LIN {X 0,Y 536.009,Z 529.66,A -85,B 0,C 180,E1 3996.244,E2 3996.244} C_VEL
LIN {X 0,Y 535.95,Z 529.66,A -85,B 0,C 180,E1 4002.513,E2 4002.513} C_VEL
LIN {X 0,Y 536.324,Z 529.982,A -85,B 0,C 180,E1 4007.164,E2 4007.164} C_VEL
LIN {X 0,Y 539.908,Z 549.024,A -85,B 0,C 180,E1 4007.547,E2 4007.547} C_VEL
LIN {X 0,Y 539.61,Z 624.102,A -85,B 0,C 180,E1 4008.663,E2 4008.663} C_VEL
LIN {X 0,Y 539.026,Z 653.248,A -85,B 0,C 180,E1 4009.753,E2 4009.753} C_VEL
LIN {X 0,Y 538.301,Z 680.399,A -85,B 0,C 180,E1 4011.48,E2 4011.48} C_VEL
LIN {X 0,Y 537.64,Z 703.617,A -85,B 0,C 180,E1 4013.748,E2 4013.748} C_VEL
LIN {X 0,Y 537.126,Z 722.234,A -85,B 0,C 180,E1 4016.46,E2 4016.46} C_VEL
LIN {X 0,Y 536.918,Z 734.161,A -85,B 0,C 180,E1 4019.136,E2 4019.136} C_VEL
LIN {X 0,Y 536.796,Z 741.628,A -85,B 0,C 180,E1 4022.073,E2 4022.073} C_VEL
LIN {X 0,Y 536.618,Z 743.988,A -85,B 0,C 180,E1 4025.051,E2 4025.051} C_VEL
LIN {X 0,Y 536.8,Z 741.206,A -85,B 0,C 180,E1 4028.077,E2 4028.077} C_VEL
LIN {X 0,Y 536.931,Z 732.797,A -85,B 0,C 180,E1 4031.143,E2 4031.143} C_VEL
LIN {X 0,Y 537.282,Z 718.414,A -85,B 0,C 180,E1 4034.107,E2 4034.107} C_VEL
LIN {X 0,Y 537.78,Z 699.357,A -85,B 0,C 180,E1 4036.65,E2 4036.65} C_VEL
LIN {X 0,Y 538.453,Z 675.808,A -85,B 0,C 180,E1 4038.779,E2 4038.779} C_VEL
LIN {X 0,Y 539.118,Z 648.555,A -85,B 0,C 180,E1 4040.382,E2 4040.382} C_VEL
LIN {X 0,Y 539.716,Z 619.376,A -85,B 0,C 180,E1 4041.356,E2 4041.356} C_VEL
LIN {X 0,Y 539.014,Z 540.519,A -85,B 0,C 180,E1 4042.509,E2 4042.509} C_VEL
LIN {X 0,Y 536.185,Z 529.66,A -85,B 0,C 180,E1 4042.825,E2 4042.825} C_VEL
LIN {X 0,Y 536.413,Z 529.66,A -85,B 0,C 180,E1 4048.387,E2 4048.387} C_VEL
LIN {X 0,Y 536.478,Z 529.66,A -85,B 0,C 180,E1 4053.224,E2 4053.224} C_VEL
LIN {X 0,Y 536.337,Z 529.66,A -85,B 0,C 180,E1 4058.086,E2 4058.086} C_VEL
LIN {X 0,Y 536.259,Z 529.66,A -85,B 0,C 180,E1 4063.009,E2 4063.009} C_VEL
LIN {X 0,Y 536.257,Z 529.66,A -85,B 0,C 180,E1 4068.03,E2 4068.03} C_VEL
LIN {X 0,Y 536.18,Z 529.66,A -85,B 0,C 180,E1 4073.203,E2 4073.203} C_VEL
LIN {X 0,Y 535.995,Z 529.66,A -85,B 0,C 180,E1 4079.218,E2 4079.218} C_VEL
LIN {X 0,Y 536.078,Z 529.66,A -85,B 0,C 180,E1 4085.28,E2 4085.28} C_VEL
LIN {X 0,Y 536.058,Z 529.66,A -85,B 0,C 180,E1 4090.53,E2 4090.53} C_VEL
LIN {X 0,Y 536.047,Z 529.66,A -85,B 0,C 180,E1 4097.046,E2 4097.046} C_VEL
LIN {X 0,Y 536.127,Z 529.66,A -85,B 0,C 180,E1 4102.006,E2 4102.006} C_VEL
LIN {X 0,Y 536.002,Z 529.66,A -85,B 0,C 180,E1 4107.661,E2 4107.661} C_VEL
LIN {X 0,Y 536.225,Z 529.66,A -85,B 0,C 180,E1 4114.224,E2 4114.224} C_VEL
LIN {X 0,Y 536.413,Z 529.66,A -85,B 0,C 180,E1 4115.573,E2 4115.573} C_VEL
LIN {X 0,Y 542.639,Z 549.532,A -85,B 0,C 180,E1 4116.157,E2 4116.157} C_VEL
LIN {X 0,Y 542.031,Z 585.577,A -85,B 0,C 180,E1 4116.981,E2 4116.981} C_VEL
LIN {X 0,Y 540.981,Z 619.2,A -85,B 0,C 180,E1 4118.415,E2 4118.415} C_VEL
LIN {X 0,Y 539.732,Z 651.158,A -85,B 0,C 180,E1 4120.501,E2 4120.501} C_VEL
LIN {X 0,Y 538.579,Z 677.691,A -85,B 0,C 180,E1 4122.945,E2 4122.945} C_VEL
LIN {X 0,Y 537.718,Z 701.766,A -85,B 0,C 180,E1 4125.994,E2 4125.994} C_VEL
LIN {X 0,Y 537.159,Z 719.995,A -85,B 0,C 180,E1 4129.228,E2 4129.228} C_VEL
LIN {X 0,Y 536.883,Z 733.409,A -85,B 0,C 180,E1 4132.732,E2 4132.732} C_VEL
LIN {X 0,Y 536.795,Z 740.394,A -85,B 0,C 180,E1 4135.732,E2 4135.732} C_VEL
LIN {X 0,Y 536.721,Z 743.474,A -85,B 0,C 180,E1 4138.387,E2 4138.387} C_VEL
LIN {X 0,Y 536.852,Z 743.419,A -85,B 0,C 180,E1 4141.609,E2 4141.609} C_VEL
LIN {X 0,Y 536.807,Z 739.198,A -85,B 0,C 180,E1 4144.835,E2 4144.835} C_VEL
LIN {X 0,Y 536.965,Z 729.095,A -85,B 0,C 180,E1 4148.482,E2 4148.482} C_VEL
LIN {X 0,Y 537.316,Z 713.592,A -85,B 0,C 180,E1 4151.951,E2 4151.951} C_VEL
LIN {X 0,Y 538.008,Z 693.827,A -85,B 0,C 180,E1 4155.035,E2 4155.035} C_VEL
LIN {X 0,Y 538.992,Z 668.188,A -85,B 0,C 180,E1 4157.934,E2 4157.934} C_VEL
LIN {X 0,Y 540.269,Z 638.35,A -85,B 0,C 180,E1 4160.343,E2 4160.343} C_VEL
LIN {X 0,Y 541.151,Z 614.891,A -85,B 0,C 180,E1 4161.718,E2 4161.718} C_VEL
LIN {X 0,Y 537.972,Z 599.622,A -85,B 0,C 180,E1 4162.578,E2 4162.578} C_VEL
LIN {X 0,Y 534.792,Z 585.979,A -85,B 0,C 180,E1 4163.245,E2 4163.245} C_VEL
LIN {X 0,Y 534.777,Z 583.899,A -85,B 0,C 180,E1 4163.316,E2 4163.316} C_VEL
LIN {X 0,Y 534.711,Z 547.853,A -85,B 0,C 180,E1 4164.152,E2 4164.152} C_VEL
LIN {X 0,Y 528.282,Z 529.66,A -85,B 0,C 180,E1 4164.754,E2 4164.754} C_VEL
LIN {X 0,Y 528.142,Z 529.66,A -85,B 0,C 180,E1 4171.003,E2 4171.003} C_VEL
LIN {X 0,Y 528.088,Z 529.66,A -85,B 0,C 180,E1 4176.871,E2 4176.871} C_VEL
LIN {X 0,Y 527.998,Z 529.66,A -85,B 0,C 180,E1 4183.303,E2 4183.303} C_VEL
LIN {X 0,Y 528.131,Z 529.66,A -85,B 0,C 180,E1 4188.917,E2 4188.917} C_VEL
LIN {X 0,Y 528.135,Z 529.66,A -85,B 0,C 180,E1 4195.15,E2 4195.15} C_VEL
LIN {X 0,Y 528.223,Z 529.66,A -85,B 0,C 180,E1 4200.411,E2 4200.411} C_VEL
LIN {X 0,Y 537.906,Z 555.81,A -85,B 0,C 180,E1 4201.345,E2 4201.345} C_VEL
LIN {X 0,Y 537.262,Z 596.398,A -85,B 0,C 180,E1 4202.129,E2 4202.129} C_VEL
LIN {X 0,Y 535.972,Z 632.816,A -85,B 0,C 180,E1 4203.464,E2 4203.464} C_VEL
LIN {X 0,Y 534.3,Z 668.478,A -85,B 0,C 180,E1 4205.493,E2 4205.493} C_VEL
LIN {X 0,Y 532.62,Z 699.844,A -85,B 0,C 180,E1 4208.007,E2 4208.007} C_VEL
LIN {X 0,Y 531.125,Z 727.043,A -85,B 0,C 180,E1 4210.93,E2 4210.93} C_VEL
LIN {X 0,Y 529.939,Z 751.815,A -85,B 0,C 180,E1 4214.518,E2 4214.518} C_VEL
LIN {X 0,Y 529.276,Z 769.655,A -85,B 0,C 180,E1 4218.072,E2 4218.072} C_VEL
LIN {X 0,Y 528.98,Z 782.685,A -85,B 0,C 180,E1 4221.801,E2 4221.801} C_VEL
LIN {X 0,Y 528.862,Z 791.191,A -85,B 0,C 180,E1 4225.91,E2 4225.91} C_VEL
LIN {X 0,Y 528.783,Z 794,A -85,B 0,C 180,E1 4230.001,E2 4230.001} C_VEL
LIN {X 0,Y 528.901,Z 791.19,A -85,B 0,C 180,E1 4234.091,E2 4234.091} C_VEL
LIN {X 0,Y 529.004,Z 782.678,A -85,B 0,C 180,E1 4238.201,E2 4238.201} C_VEL
LIN {X 0,Y 529.253,Z 769.649,A -85,B 0,C 180,E1 4241.93,E2 4241.93} C_VEL
LIN {X 0,Y 529.975,Z 750.599,A -85,B 0,C 180,E1 4245.694,E2 4245.694} C_VEL
LIN {X 0,Y 531.118,Z 727.031,A -85,B 0,C 180,E1 4249.071,E2 4249.071} C_VEL
LIN {X 0,Y 532.597,Z 699.86,A -85,B 0,C 180,E1 4251.992,E2 4251.992} C_VEL
LIN {X 0,Y 534.276,Z 668.46,A -85,B 0,C 180,E1 4254.509,E2 4254.509} C_VEL
LIN {X 0,Y 535.917,Z 633.307,A -85,B 0,C 180,E1 4256.516,E2 4256.516} C_VEL
LIN {X 0,Y 537.203,Z 596.71,A -85,B 0,C 180,E1 4257.866,E2 4257.866} C_VEL
LIN {X 0,Y 537.47,Z 553.409,A -85,B 0,C 180,E1 4258.717,E2 4258.717} C_VEL
LIN {X 0,Y 528.217,Z 529.66,A -85,B 0,C 180,E1 4259.593,E2 4259.593} C_VEL
LIN {X 0,Y 528.124,Z 529.66,A -85,B 0,C 180,E1 4264.852,E2 4264.852} C_VEL
LIN {X 0,Y 528.156,Z 529.66,A -85,B 0,C 180,E1 4269.523,E2 4269.523} C_VEL
LIN {X 0,Y 528.089,Z 529.66,A -85,B 0,C 180,E1 4275.592,E2 4275.592} C_VEL
LIN {X 0,Y 528.134,Z 529.66,A -85,B 0,C 180,E1 4281.057,E2 4281.057} C_VEL
LIN {X 0,Y 528.12,Z 529.66,A -85,B 0,C 180,E1 4287.123,E2 4287.123} C_VEL
LIN {X 0,Y 528.196,Z 529.66,A -85,B 0,C 180,E1 4292.803,E2 4292.803} C_VEL
LIN {X 0,Y 528.328,Z 529.66,A -85,B 0,C 180,E1 4298.207,E2 4298.207} C_VEL
LIN {X 0,Y 528.423,Z 529.66,A -85,B 0,C 180,E1 4303.41,E2 4303.41} C_VEL
LIN {X 0,Y 528.47,Z 529.66,A -85,B 0,C 180,E1 4310.138,E2 4310.138} C_VEL
LIN {X 0,Y 528.582,Z 529.66,A -85,B 0,C 180,E1 4315.089,E2 4315.089} C_VEL
LIN {X 0,Y 528.64,Z 529.66,A -85,B 0,C 180,E1 4320.002,E2 4320.002} C_VEL
LIN {X 0,Y 528.61,Z 529.66,A -85,B 0,C 180,E1 4324.915,E2 4324.915} C_VEL
LIN {X 0,Y 528.501,Z 529.66,A -85,B 0,C 180,E1 4329.866,E2 4329.866} C_VEL
LIN {X 0,Y 528.464,Z 529.66,A -85,B 0,C 180,E1 4334.894,E2 4334.894} C_VEL
LIN {X 0,Y 528.375,Z 529.66,A -85,B 0,C 180,E1 4340.044,E2 4340.044} C_VEL
LIN {X 0,Y 528.202,Z 529.66,A -85,B 0,C 180,E1 4345.376,E2 4345.376} C_VEL
LIN {X 0,Y 528.141,Z 529.66,A -85,B 0,C 180,E1 4351,E2 4351} C_VEL
LIN {X 0,Y 528.069,Z 529.66,A -85,B 0,C 180,E1 4356.878,E2 4356.878} C_VEL
LIN {X 0,Y 528.014,Z 529.66,A -85,B 0,C 180,E1 4363.308,E2 4363.308} C_VEL
LIN {X 0,Y 528.365,Z 529.66,A -85,B 0,C 180,E1 4366.859,E2 4366.859} C_VEL
LIN {X 0,Y 532.147,Z 547.399,A -85,B 0,C 180,E1 4367.261,E2 4367.261} C_VEL
LIN {X 0,Y 532.046,Z 624.585,A -85,B 0,C 180,E1 4368.431,E2 4368.431} C_VEL
LIN {X 0,Y 531.393,Z 653.619,A -85,B 0,C 180,E1 4369.532,E2 4369.532} C_VEL
LIN {X 0,Y 530.6,Z 680.452,A -85,B 0,C 180,E1 4371.268,E2 4371.268} C_VEL
LIN {X 0,Y 529.858,Z 702.607,A -85,B 0,C 180,E1 4373.452,E2 4373.452} C_VEL
LIN {X 0,Y 529.328,Z 720.972,A -85,B 0,C 180,E1 4376.111,E2 4376.111} C_VEL
LIN {X 0,Y 529.026,Z 734.353,A -85,B 0,C 180,E1 4379.107,E2 4379.107} C_VEL
LIN {X 0,Y 528.89,Z 741.859,A -85,B 0,C 180,E1 4382.19,E2 4382.19} C_VEL
LIN {X 0,Y 528.738,Z 743.945,A -85,B 0,C 180,E1 4384.653,E2 4384.653} C_VEL
LIN {X 0,Y 528.842,Z 741.854,A -85,B 0,C 180,E1 4387.729,E2 4387.729} C_VEL
LIN {X 0,Y 529.034,Z 734.88,A -85,B 0,C 180,E1 4390.639,E2 4390.639} C_VEL
LIN {X 0,Y 529.289,Z 721.837,A -85,B 0,C 180,E1 4393.647,E2 4393.647} C_VEL
LIN {X 0,Y 529.88,Z 703.234,A -85,B 0,C 180,E1 4396.38,E2 4396.38} C_VEL
LIN {X 0,Y 530.598,Z 680.819,A -85,B 0,C 180,E1 4398.611,E2 4398.611} C_VEL
LIN {X 0,Y 531.409,Z 654.236,A -85,B 0,C 180,E1 4400.344,E2 4400.344} C_VEL
LIN {X 0,Y 531.994,Z 626.187,A -85,B 0,C 180,E1 4401.435,E2 4401.435} C_VEL
LIN {X 0,Y 532.245,Z 567.67,A -85,B 0,C 180,E1 4402.364,E2 4402.364} C_VEL
LIN {X 0,Y 531.319,Z 541.394,A -85,B 0,C 180,E1 4402.761,E2 4402.761} C_VEL
LIN {X 0,Y 528.288,Z 529.66,A -85,B 0,C 180,E1 4403.116,E2 4403.116} C_VEL
LIN {X 0,Y 528.523,Z 529.66,A -85,B 0,C 180,E1 4408.363,E2 4408.363} C_VEL
LIN {X 0,Y 528.585,Z 529.66,A -85,B 0,C 180,E1 4413.272,E2 4413.272} C_VEL
LIN {X 0,Y 528.44,Z 529.66,A -85,B 0,C 180,E1 4418.208,E2 4418.208} C_VEL
LIN {X 0,Y 528.313,Z 529.66,A -85,B 0,C 180,E1 4423.797,E2 4423.797} C_VEL
LIN {X 0,Y 528.374,Z 529.66,A -85,B 0,C 180,E1 4429.528,E2 4429.528} C_VEL
LIN {X 0,Y 528.205,Z 529.66,A -85,B 0,C 180,E1 4435.373,E2 4435.373} C_VEL
LIN {X 0,Y 528.09,Z 529.66,A -85,B 0,C 180,E1 4440.989,E2 4440.989} C_VEL
LIN {X 0,Y 528.255,Z 529.66,A -85,B 0,C 180,E1 4446.883,E2 4446.883} C_VEL
LIN {X 0,Y 528.03,Z 529.66,A -85,B 0,C 180,E1 4453.303,E2 4453.303} C_VEL
LIN {X 0,Y 528.103,Z 529.66,A -85,B 0,C 180,E1 4458.911,E2 4458.911} C_VEL
LIN {X 0,Y 528.069,Z 529.66,A -85,B 0,C 180,E1 4465.142,E2 4465.142} C_VEL
LIN {X 0,Y 528.155,Z 529.66,A -85,B 0,C 180,E1 4470.939,E2 4470.939} C_VEL
LIN {X 0,Y 528.447,Z 529.66,A -85,B 0,C 180,E1 4475.163,E2 4475.163} C_VEL
LIN {X 0,Y 535.451,Z 551.381,A -85,B 0,C 180,E1 4475.846,E2 4475.846} C_VEL
LIN {X 0,Y 534.695,Z 586.678,A -85,B 0,C 180,E1 4476.686,E2 4476.686} C_VEL
LIN {X 0,Y 533.505,Z 621.104,A -85,B 0,C 180,E1 4478.206,E2 4478.206} C_VEL
LIN {X 0,Y 532.146,Z 652.485,A -85,B 0,C 180,E1 4480.32,E2 4480.32} C_VEL
LIN {X 0,Y 530.818,Z 680.078,A -85,B 0,C 180,E1 4482.955,E2 4482.955} C_VEL
LIN {X 0,Y 529.842,Z 704.046,A -85,B 0,C 180,E1 4486.136,E2 4486.136} C_VEL
LIN {X 0,Y 529.258,Z 721.344,A -85,B 0,C 180,E1 4489.356,E2 4489.356} C_VEL
LIN {X 0,Y 528.995,Z 734.551,A -85,B 0,C 180,E1 4493.035,E2 4493.035} C_VEL
LIN {X 0,Y 528.917,Z 741.947,A -85,B 0,C 180,E1 4496.727,E2 4496.727} C_VEL
LIN {X 0,Y 528.806,Z 743.997,A -85,B 0,C 180,E1 4499.998,E2 4499.998} C_VEL
LIN {X 0,Y 528.916,Z 741.843,A -85,B 0,C 180,E1 4503.269,E2 4503.269} C_VEL
LIN {X 0,Y 529.011,Z 734.311,A -85,B 0,C 180,E1 4506.961,E2 4506.961} C_VEL
LIN {X 0,Y 529.356,Z 720.626,A -85,B 0,C 180,E1 4510.708,E2 4510.708} C_VEL
LIN {X 0,Y 530.015,Z 701.179,A -85,B 0,C 180,E1 4514.211,E2 4514.211} C_VEL
LIN {X 0,Y 530.959,Z 677.649,A -85,B 0,C 180,E1 4517.221,E2 4517.221} C_VEL
LIN {X 0,Y 532.276,Z 650.083,A -85,B 0,C 180,E1 4519.778,E2 4519.778} C_VEL
LIN {X 0,Y 533.553,Z 619.596,A -85,B 0,C 180,E1 4521.787,E2 4521.787} C_VEL
LIN {X 0,Y 534.723,Z 585.396,A -85,B 0,C 180,E1 4523.268,E2 4523.268} C_VEL
LIN {X 0,Y 534.777,Z 583.899,A -85,B 0,C 180,E1 4523.316,E2 4523.316} C_VEL
LIN {X 0,Y 533.025,Z 567.224,A -85,B 0,C 180,E1 4523.874,E2 4523.874} C_VEL
LIN {X 0,Y 527.988,Z 551.07,A -85,B 0,C 180,E1 4524.432,E2 4524.432} C_VEL
LIN {X 0,Y 520.329,Z 529.66,A -85,B 0,C 180,E1 4525.219,E2 4525.219} C_VEL
LIN {X 0,Y 520.224,Z 529.66,A -85,B 0,C 180,E1 4531.471,E2 4531.471} C_VEL
LIN {X 0,Y 520.089,Z 529.66,A -85,B 0,C 180,E1 4537.535,E2 4537.535} C_VEL
LIN {X 0,Y 520.093,Z 529.66,A -85,B 0,C 180,E1 4543.503,E2 4543.503} C_VEL
LIN {X 0,Y 520.228,Z 529.66,A -85,B 0,C 180,E1 4548.948,E2 4548.948} C_VEL
LIN {X 0,Y 520.185,Z 529.66,A -85,B 0,C 180,E1 4554.538,E2 4554.538} C_VEL
LIN {X 0,Y 520.314,Z 529.66,A -85,B 0,C 180,E1 4560.082,E2 4560.082} C_VEL
LIN {X 0,Y 530.949,Z 556.615,A -85,B 0,C 180,E1 4560.953,E2 4560.953} C_VEL
LIN {X 0,Y 530.248,Z 597.126,A -85,B 0,C 180,E1 4561.748,E2 4561.748} C_VEL
LIN {X 0,Y 528.822,Z 632.931,A -85,B 0,C 180,E1 4563.082,E2 4563.082} C_VEL
LIN {X 0,Y 526.98,Z 668.474,A -85,B 0,C 180,E1 4565.13,E2 4565.13} C_VEL
LIN {X 0,Y 525.142,Z 700.197,A -85,B 0,C 180,E1 4567.712,E2 4567.712} C_VEL
LIN {X 0,Y 523.41,Z 728.787,A -85,B 0,C 180,E1 4570.857,E2 4570.857} C_VEL
LIN {X 0,Y 522.103,Z 753.018,A -85,B 0,C 180,E1 4574.494,E2 4574.494} C_VEL
LIN {X 0,Y 521.367,Z 771.385,A -85,B 0,C 180,E1 4578.312,E2 4578.312} C_VEL
LIN {X 0,Y 521.057,Z 783.828,A -85,B 0,C 180,E1 4582.094,E2 4582.094} C_VEL
LIN {X 0,Y 520.959,Z 791.192,A -85,B 0,C 180,E1 4585.848,E2 4585.848} C_VEL
LIN {X 0,Y 520.889,Z 794,A -85,B 0,C 180,E1 4590.001,E2 4590.001} C_VEL
LIN {X 0,Y 520.994,Z 791.191,A -85,B 0,C 180,E1 4594.153,E2 4594.153} C_VEL
LIN {X 0,Y 521.115,Z 782.678,A -85,B 0,C 180,E1 4598.326,E2 4598.326} C_VEL
LIN {X 0,Y 521.409,Z 769.649,A -85,B 0,C 180,E1 4602.113,E2 4602.113} C_VEL
LIN {X 0,Y 522.207,Z 750.6,A -85,B 0,C 180,E1 4605.934,E2 4605.934} C_VEL
LIN {X 0,Y 523.475,Z 727.031,A -85,B 0,C 180,E1 4609.361,E2 4609.361} C_VEL
LIN {X 0,Y 525.23,Z 698.46,A -85,B 0,C 180,E1 4612.453,E2 4612.453} C_VEL
LIN {X 0,Y 527.094,Z 666.926,A -85,B 0,C 180,E1 4614.979,E2 4614.979} C_VEL
LIN {X 0,Y 528.927,Z 631.177,A -85,B 0,C 180,E1 4616.995,E2 4616.995} C_VEL
LIN {X 0,Y 530.246,Z 596.382,A -85,B 0,C 180,E1 4618.273,E2 4618.273} C_VEL
LIN {X 0,Y 530.592,Z 555.708,A -85,B 0,C 180,E1 4619.079,E2 4619.079} C_VEL
LIN {X 0,Y 520.275,Z 529.66,A -85,B 0,C 180,E1 4620.061,E2 4620.061} C_VEL
LIN {X 0,Y 520.216,Z 529.66,A -85,B 0,C 180,E1 4625.694,E2 4625.694} C_VEL
LIN {X 0,Y 520.191,Z 529.66,A -85,B 0,C 180,E1 4631.047,E2 4631.047} C_VEL
LIN {X 0,Y 520.173,Z 529.66,A -85,B 0,C 180,E1 4636.489,E2 4636.489} C_VEL
LIN {X 0,Y 520.224,Z 529.66,A -85,B 0,C 180,E1 4642.476,E2 4642.476} C_VEL
LIN {X 0,Y 520.192,Z 529.66,A -85,B 0,C 180,E1 4648.526,E2 4648.526} C_VEL
LIN {X 0,Y 520.295,Z 529.66,A -85,B 0,C 180,E1 4654.215,E2 4654.215} C_VEL
LIN {X 0,Y 520.449,Z 529.66,A -85,B 0,C 180,E1 4659.642,E2 4659.642} C_VEL
LIN {X 0,Y 520.358,Z 529.66,A -85,B 0,C 180,E1 4664.874,E2 4664.874} C_VEL
LIN {X 0,Y 520.585,Z 529.66,A -85,B 0,C 180,E1 4670.248,E2 4670.248} C_VEL
LIN {X 0,Y 520.677,Z 529.66,A -85,B 0,C 180,E1 4675.014,E2 4675.014} C_VEL
LIN {X 0,Y 520.752,Z 529.66,A -85,B 0,C 180,E1 4680.002,E2 4680.002} C_VEL
LIN {X 0,Y 520.695,Z 529.66,A -85,B 0,C 180,E1 4684.99,E2 4684.99} C_VEL
LIN {X 0,Y 520.576,Z 529.66,A -85,B 0,C 180,E1 4690.018,E2 4690.018} C_VEL
LIN {X 0,Y 520.53,Z 529.66,A -85,B 0,C 180,E1 4695.126,E2 4695.126} C_VEL
LIN {X 0,Y 520.431,Z 529.66,A -85,B 0,C 180,E1 4700.363,E2 4700.363} C_VEL
LIN {X 0,Y 520.236,Z 529.66,A -85,B 0,C 180,E1 4705.948,E2 4705.948} C_VEL
LIN {X 0,Y 520.212,Z 529.66,A -85,B 0,C 180,E1 4711.477,E2 4711.477} C_VEL
LIN {X 0,Y 520.063,Z 529.66,A -85,B 0,C 180,E1 4717.543,E2 4717.543} C_VEL
LIN {X 0,Y 520.112,Z 529.66,A -85,B 0,C 180,E1 4723.503,E2 4723.503} C_VEL
LIN {X 0,Y 520.402,Z 529.66,A -85,B 0,C 180,E1 4726.575,E2 4726.575} C_VEL
LIN {X 0,Y 524.617,Z 548.131,A -85,B 0,C 180,E1 4727.007,E2 4727.007} C_VEL
LIN {X 0,Y 524.49,Z 625.285,A -85,B 0,C 180,E1 4728.198,E2 4728.198} C_VEL
LIN {X 0,Y 523.813,Z 653.189,A -85,B 0,C 180,E1 4729.263,E2 4729.263} C_VEL
LIN {X 0,Y 522.986,Z 679.327,A -85,B 0,C 180,E1 4730.947,E2 4730.947} C_VEL
LIN {X 0,Y 522.129,Z 702.433,A -85,B 0,C 180,E1 4733.211,E2 4733.211} C_VEL
LIN {X 0,Y 521.522,Z 721.035,A -85,B 0,C 180,E1 4735.943,E2 4735.943} C_VEL
LIN {X 0,Y 521.159,Z 734.536,A -85,B 0,C 180,E1 4739.042,E2 4739.042} C_VEL
LIN {X 0,Y 520.978,Z 742.239,A -85,B 0,C 180,E1 4742.39,E2 4742.39} C_VEL
LIN {X 0,Y 520.814,Z 743.86,A -85,B 0,C 180,E1 4744.239,E2 4744.239} C_VEL
LIN {X 0,Y 520.823,Z 743.638,A -85,B 0,C 180,E1 4746.069,E2 4746.069} C_VEL
LIN {X 0,Y 521.069,Z 740.017,A -85,B 0,C 180,E1 4748.815,E2 4748.815} C_VEL
LIN {X 0,Y 521.235,Z 731.187,A -85,B 0,C 180,E1 4751.796,E2 4751.796} C_VEL
LIN {X 0,Y 521.667,Z 716.778,A -85,B 0,C 180,E1 4754.695,E2 4754.695} C_VEL
LIN {X 0,Y 522.31,Z 697.392,A -85,B 0,C 180,E1 4757.273,E2 4757.273} C_VEL
LIN {X 0,Y 523.161,Z 674.318,A -85,B 0,C 180,E1 4759.345,E2 4759.345} C_VEL
LIN {X 0,Y 523.975,Z 647.028,A -85,B 0,C 180,E1 4760.938,E2 4760.938} C_VEL
LIN {X 0,Y 524.556,Z 617.97,A -85,B 0,C 180,E1 4761.886,E2 4761.886} C_VEL
LIN {X 0,Y 523.89,Z 543.047,A -85,B 0,C 180,E1 4763,E2 4763} C_VEL
LIN {X 0,Y 520.363,Z 529.66,A -85,B 0,C 180,E1 4763.338,E2 4763.338} C_VEL
LIN {X 0,Y 520.647,Z 529.66,A -85,B 0,C 180,E1 4768.338,E2 4768.338} C_VEL
LIN {X 0,Y 520.681,Z 529.66,A -85,B 0,C 180,E1 4773.322,E2 4773.322} C_VEL
LIN {X 0,Y 520.528,Z 529.66,A -85,B 0,C 180,E1 4778.334,E2 4778.334} C_VEL
LIN {X 0,Y 520.452,Z 529.66,A -85,B 0,C 180,E1 4783.411,E2 4783.411} C_VEL
LIN {X 0,Y 520.433,Z 529.66,A -85,B 0,C 180,E1 4788.598,E2 4788.598} C_VEL
LIN {X 0,Y 520.314,Z 529.66,A -85,B 0,C 180,E1 4793.954,E2 4793.954} C_VEL
LIN {X 0,Y 520.179,Z 529.66,A -85,B 0,C 180,E1 4799.547,E2 4799.547} C_VEL
LIN {X 0,Y 520.231,Z 529.66,A -85,B 0,C 180,E1 4805.688,E2 4805.688} C_VEL
LIN {X 0,Y 520.168,Z 529.66,A -85,B 0,C 180,E1 4811.037,E2 4811.037} C_VEL
LIN {X 0,Y 520.184,Z 529.66,A -85,B 0,C 180,E1 4816.486,E2 4816.486} C_VEL
LIN {X 0,Y 520.171,Z 529.66,A -85,B 0,C 180,E1 4822.466,E2 4822.466} C_VEL
LIN {X 0,Y 520.164,Z 529.66,A -85,B 0,C 180,E1 4828.519,E2 4828.519} C_VEL
LIN {X 0,Y 520.475,Z 529.66,A -85,B 0,C 180,E1 4834.777,E2 4834.777} C_VEL
LIN {X 0,Y 528.239,Z 553.901,A -85,B 0,C 180,E1 4835.538,E2 4835.538} C_VEL
LIN {X 0,Y 527.355,Z 589.315,A -85,B 0,C 180,E1 4836.439,E2 4836.439} C_VEL
LIN {X 0,Y 526.049,Z 623.008,A -85,B 0,C 180,E1 4837.992,E2 4837.992} C_VEL
LIN {X 0,Y 524.544,Z 653.801,A -85,B 0,C 180,E1 4840.132,E2 4840.132} C_VEL
LIN {X 0,Y 523.068,Z 682.108,A -85,B 0,C 180,E1 4842.927,E2 4842.927} C_VEL
LIN {X 0,Y 522.05,Z 704.573,A -85,B 0,C 180,E1 4846.01,E2 4846.01} C_VEL
LIN {X 0,Y 521.357,Z 722.985,A -85,B 0,C 180,E1 4849.587,E2 4849.587} C_VEL
LIN {X 0,Y 521.127,Z 734.55,A -85,B 0,C 180,E1 4852.929,E2 4852.929} C_VEL
LIN {X 0,Y 521.014,Z 741.943,A -85,B 0,C 180,E1 4856.677,E2 4856.677} C_VEL
LIN {X 0,Y 520.912,Z 743.997,A -85,B 0,C 180,E1 4859.998,E2 4859.998} C_VEL
LIN {X 0,Y 521.014,Z 741.841,A -85,B 0,C 180,E1 4863.318,E2 4863.318} C_VEL
LIN {X 0,Y 521.147,Z 734.314,A -85,B 0,C 180,E1 4867.066,E2 4867.066} C_VEL
LIN {X 0,Y 521.516,Z 720.605,A -85,B 0,C 180,E1 4870.877,E2 4870.877} C_VEL
LIN {X 0,Y 522.228,Z 701.986,A -85,B 0,C 180,E1 4874.306,E2 4874.306} C_VEL
LIN {X 0,Y 523.249,Z 678.576,A -85,B 0,C 180,E1 4877.379,E2 4877.379} C_VEL
LIN {X 0,Y 524.676,Z 651.439,A -85,B 0,C 180,E1 4879.968,E2 4879.968} C_VEL
LIN {X 0,Y 526.176,Z 619.604,A -85,B 0,C 180,E1 4882.108,E2 4882.108} C_VEL
LIN {X 0,Y 527.456,Z 585.415,A -85,B 0,C 180,E1 4883.608,E2 4883.608} C_VEL
LIN {X 0,Y 527.988,Z 551.07,A -85,B 0,C 180,E1 4884.432,E2 4884.432} C_VEL
LIN {X 0,Y 520.994,Z 542.646,A -85,B 0,C 180,E1 4884.915,E2 4884.915} C_VEL
LIN {X 0,Y 513.747,Z 534.323,A -85,B 0,C 180,E1 4885.406,E2 4885.406} C_VEL
LIN {X 0,Y 512.392,Z 529.66,A -85,B 0,C 180,E1 4885.606,E2 4885.606} C_VEL
LIN {X 0,Y 512.331,Z 529.66,A -85,B 0,C 180,E1 4892.013,E2 4892.013} C_VEL
LIN {X 0,Y 512.185,Z 529.66,A -85,B 0,C 180,E1 4898.218,E2 4898.218} C_VEL
LIN {X 0,Y 512.196,Z 529.66,A -85,B 0,C 180,E1 4905.004,E2 4905.004} C_VEL
LIN {X 0,Y 512.323,Z 529.66,A -85,B 0,C 180,E1 4909.974,E2 4909.974} C_VEL
LIN {X 0,Y 512.241,Z 529.66,A -85,B 0,C 180,E1 4915.965,E2 4915.965} C_VEL
LIN {X 0,Y 512.368,Z 529.66,A -85,B 0,C 180,E1 4919.726,E2 4919.726} C_VEL
LIN {X 0,Y 523.614,Z 558.863,A -85,B 0,C 180,E1 4920.666,E2 4920.666} C_VEL
LIN {X 0,Y 522.963,Z 599.981,A -85,B 0,C 180,E1 4921.483,E2 4921.483} C_VEL
LIN {X 0,Y 521.555,Z 636.941,A -85,B 0,C 180,E1 4922.891,E2 4922.891} C_VEL
LIN {X 0,Y 519.617,Z 670.002,A -85,B 0,C 180,E1 4924.868,E2 4924.868} C_VEL
LIN {X 0,Y 517.639,Z 700.696,A -85,B 0,C 180,E1 4927.42,E2 4927.42} C_VEL
LIN {X 0,Y 515.791,Z 728.787,A -85,B 0,C 180,E1 4930.563,E2 4930.563} C_VEL
LIN {X 0,Y 514.357,Z 753.017,A -85,B 0,C 180,E1 4934.255,E2 4934.255} C_VEL
LIN {X 0,Y 513.523,Z 771.385,A -85,B 0,C 180,E1 4938.131,E2 4938.131} C_VEL
LIN {X 0,Y 513.197,Z 783.828,A -85,B 0,C 180,E1 4941.972,E2 4941.972} C_VEL
LIN {X 0,Y 513.057,Z 791.192,A -85,B 0,C 180,E1 4945.784,E2 4945.784} C_VEL
LIN {X 0,Y 512.994,Z 794,A -85,B 0,C 180,E1 4950.001,E2 4950.001} C_VEL
LIN {X 0,Y 513.087,Z 791.191,A -85,B 0,C 180,E1 4954.217,E2 4954.217} C_VEL
LIN {X 0,Y 513.245,Z 782.678,A -85,B 0,C 180,E1 4958.454,E2 4958.454} C_VEL
LIN {X 0,Y 513.561,Z 769.648,A -85,B 0,C 180,E1 4962.3,E2 4962.3} C_VEL
LIN {X 0,Y 514.456,Z 750.601,A -85,B 0,C 180,E1 4966.18,E2 4966.18} C_VEL
LIN {X 0,Y 515.853,Z 727.03,A -85,B 0,C 180,E1 4969.659,E2 4969.659} C_VEL
LIN {X 0,Y 517.708,Z 699.2,A -85,B 0,C 180,E1 4972.724,E2 4972.724} C_VEL
LIN {X 0,Y 519.823,Z 666.922,A -85,B 0,C 180,E1 4975.353,E2 4975.353} C_VEL
LIN {X 0,Y 521.766,Z 632.261,A -85,B 0,C 180,E1 4977.331,E2 4977.331} C_VEL
LIN {X 0,Y 523.111,Z 596.014,A -85,B 0,C 180,E1 4978.651,E2 4978.651} C_VEL
LIN {X 0,Y 523.218,Z 557.302,A -85,B 0,C 180,E1 4979.433,E2 4979.433} C_VEL
LIN {X 0,Y 512.35,Z 529.66,A -85,B 0,C 180,E1 4980.517,E2 4980.517} C_VEL
LIN {X 0,Y 512.337,Z 529.66,A -85,B 0,C 180,E1 4987.327,E2 4987.327} C_VEL
LIN {X 0,Y 512.18,Z 529.66,A -85,B 0,C 180,E1 4992.66,E2 4992.66} C_VEL
LIN {X 0,Y 512.246,Z 529.66,A -85,B 0,C 180,E1 4997.432,E2 4997.432} C_VEL
LIN {X 0,Y 512.294,Z 529.66,A -85,B 0,C 180,E1 5002.685,E2 5002.685} C_VEL
LIN {X 0,Y 512.29,Z 529.66,A -85,B 0,C 180,E1 5008.675,E2 5008.675} C_VEL
LIN {X 0,Y 512.366,Z 529.66,A -85,B 0,C 180,E1 5013.786,E2 5013.786} C_VEL
LIN {X 0,Y 512.541,Z 529.66,A -85,B 0,C 180,E1 5019.314,E2 5019.314} C_VEL
LIN {X 0,Y 512.451,Z 529.66,A -85,B 0,C 180,E1 5024.634,E2 5024.634} C_VEL
LIN {X 0,Y 512.625,Z 529.66,A -85,B 0,C 180,E1 5029.83,E2 5029.83} C_VEL
LIN {X 0,Y 512.796,Z 529.66,A -85,B 0,C 180,E1 5034.938,E2 5034.938} C_VEL
LIN {X 0,Y 512.858,Z 529.66,A -85,B 0,C 180,E1 5040.002,E2 5040.002} C_VEL
LIN {X 0,Y 512.806,Z 529.66,A -85,B 0,C 180,E1 5045.067,E2 5045.067} C_VEL
LIN {X 0,Y 512.654,Z 529.66,A -85,B 0,C 180,E1 5050.174,E2 5050.174} C_VEL
LIN {X 0,Y 512.596,Z 529.66,A -85,B 0,C 180,E1 5055.366,E2 5055.366} C_VEL
LIN {X 0,Y 512.528,Z 529.66,A -85,B 0,C 180,E1 5060.692,E2 5060.692} C_VEL
LIN {X 0,Y 512.318,Z 529.66,A -85,B 0,C 180,E1 5066.222,E2 5066.222} C_VEL
LIN {X 0,Y 512.289,Z 529.66,A -85,B 0,C 180,E1 5072.022,E2 5072.022} C_VEL
LIN {X 0,Y 512.141,Z 529.66,A -85,B 0,C 180,E1 5078.227,E2 5078.227} C_VEL
LIN {X 0,Y 512.286,Z 529.66,A -85,B 0,C 180,E1 5085.012,E2 5085.012} C_VEL
LIN {X 0,Y 512.461,Z 529.66,A -85,B 0,C 180,E1 5086.279,E2 5086.279} C_VEL
LIN {X 0,Y 517.212,Z 549.714,A -85,B 0,C 180,E1 5086.763,E2 5086.763} C_VEL
LIN {X 0,Y 516.944,Z 625.567,A -85,B 0,C 180,E1 5087.947,E2 5087.947} C_VEL
LIN {X 0,Y 516.191,Z 654.507,A -85,B 0,C 180,E1 5089.079,E2 5089.079} C_VEL
LIN {X 0,Y 515.274,Z 681.166,A -85,B 0,C 180,E1 5090.854,E2 5090.854} C_VEL
LIN {X 0,Y 514.331,Z 703.878,A -85,B 0,C 180,E1 5093.166,E2 5093.166} C_VEL
LIN {X 0,Y 513.681,Z 721.845,A -85,B 0,C 180,E1 5095.883,E2 5095.883} C_VEL
LIN {X 0,Y 513.331,Z 734.632,A -85,B 0,C 180,E1 5098.861,E2 5098.861} C_VEL
LIN {X 0,Y 513.122,Z 742.015,A -85,B 0,C 180,E1 5101.931,E2 5101.931} C_VEL
LIN {X 0,Y 512.975,Z 744.007,A -85,B 0,C 180,E1 5103.816,E2 5103.816} C_VEL
LIN {X 0,Y 512.928,Z 744.192,A -85,B 0,C 180,E1 5105.786,E2 5105.786} C_VEL
LIN {X 0,Y 513.16,Z 741.08,A -85,B 0,C 180,E1 5108.511,E2 5108.511} C_VEL
LIN {X 0,Y 513.364,Z 732.758,A -85,B 0,C 180,E1 5111.579,E2 5111.579} C_VEL
LIN {X 0,Y 513.806,Z 719.466,A -85,B 0,C 180,E1 5114.455,E2 5114.455} C_VEL
LIN {X 0,Y 514.467,Z 701.085,A -85,B 0,C 180,E1 5117.076,E2 5117.076} C_VEL
LIN {X 0,Y 515.347,Z 678.713,A -85,B 0,C 180,E1 5119.248,E2 5119.248} C_VEL
LIN {X 0,Y 516.287,Z 651.95,A -85,B 0,C 180,E1 5120.961,E2 5120.961} C_VEL
LIN {X 0,Y 516.924,Z 623.623,A -85,B 0,C 180,E1 5122.011,E2 5122.011} C_VEL
LIN {X 0,Y 516.676,Z 545.49,A -85,B 0,C 180,E1 5123.227,E2 5123.227} C_VEL
LIN {X 0,Y 512.476,Z 529.66,A -85,B 0,C 180,E1 5123.679,E2 5123.679} C_VEL
LIN {X 0,Y 512.747,Z 529.66,A -85,B 0,C 180,E1 5128.313,E2 5128.313} C_VEL
LIN {X 0,Y 512.784,Z 529.66,A -85,B 0,C 180,E1 5133.373,E2 5133.373} C_VEL
LIN {X 0,Y 512.62,Z 529.66,A -85,B 0,C 180,E1 5138.463,E2 5138.463} C_VEL
LIN {X 0,Y 512.533,Z 529.66,A -85,B 0,C 180,E1 5143.686,E2 5143.686} C_VEL
LIN {X 0,Y 512.488,Z 529.66,A -85,B 0,C 180,E1 5149.567,E2 5149.567} C_VEL
LIN {X 0,Y 512.363,Z 529.66,A -85,B 0,C 180,E1 5154.35,E2 5154.35} C_VEL
LIN {X 0,Y 512.218,Z 529.66,A -85,B 0,C 180,E1 5160.053,E2 5160.053} C_VEL
LIN {X 0,Y 512.314,Z 529.66,A -85,B 0,C 180,E1 5166.091,E2 5166.091} C_VEL
LIN {X 0,Y 512.279,Z 529.66,A -85,B 0,C 180,E1 5170.393,E2 5170.393} C_VEL
LIN {X 0,Y 512.225,Z 529.66,A -85,B 0,C 180,E1 5175.004,E2 5175.004} C_VEL
LIN {X 0,Y 512.298,Z 529.66,A -85,B 0,C 180,E1 5179.981,E2 5179.981} C_VEL
LIN {X 0,Y 512.169,Z 529.66,A -85,B 0,C 180,E1 5185.956,E2 5185.956} C_VEL
LIN {X 0,Y 512.336,Z 529.66,A -85,B 0,C 180,E1 5192.077,E2 5192.077} C_VEL
LIN {X 0,Y 512.562,Z 530.317,A -85,B 0,C 180,E1 5194.378,E2 5194.378} C_VEL
LIN {X 0,Y 521.05,Z 554.978,A -85,B 0,C 180,E1 5195.198,E2 5195.198} C_VEL
LIN {X 0,Y 520.085,Z 589.287,A -85,B 0,C 180,E1 5196.089,E2 5196.089} C_VEL
LIN {X 0,Y 518.746,Z 621.318,A -85,B 0,C 180,E1 5197.567,E2 5197.567} C_VEL
LIN {X 0,Y 517.096,Z 652.461,A -85,B 0,C 180,E1 5199.722,E2 5199.722} C_VEL
LIN {X 0,Y 515.51,Z 680.237,A -85,B 0,C 180,E1 5202.452,E2 5202.452} C_VEL
LIN {X 0,Y 514.312,Z 703.727,A -85,B 0,C 180,E1 5205.657,E2 5205.657} C_VEL
LIN {X 0,Y 513.514,Z 722.463,A -85,B 0,C 180,E1 5209.3,E2 5209.3} C_VEL
LIN {X 0,Y 513.261,Z 734.546,A -85,B 0,C 180,E1 5212.82,E2 5212.82} C_VEL
LIN {X 0,Y 513.129,Z 741.939,A -85,B 0,C 180,E1 5216.626,E2 5216.626} C_VEL
LIN {X 0,Y 513.014,Z 743.998,A -85,B 0,C 180,E1 5219.998,E2 5219.998} C_VEL
LIN {X 0,Y 513.13,Z 741.838,A -85,B 0,C 180,E1 5223.37,E2 5223.37} C_VEL
LIN {X 0,Y 513.282,Z 734.317,A -85,B 0,C 180,E1 5227.175,E2 5227.175} C_VEL
LIN {X 0,Y 513.653,Z 720.789,A -85,B 0,C 180,E1 5231.006,E2 5231.006} C_VEL
LIN {X 0,Y 514.45,Z 701.864,A -85,B 0,C 180,E1 5234.546,E2 5234.546} C_VEL
LIN {X 0,Y 515.6,Z 678.228,A -85,B 0,C 180,E1 5237.686,E2 5237.686} C_VEL
LIN {X 0,Y 517.214,Z 650.098,A -85,B 0,C 180,E1 5240.38,E2 5240.38} C_VEL
LIN {X 0,Y 518.822,Z 619.744,A -85,B 0,C 180,E1 5242.431,E2 5242.431} C_VEL
LIN {X 0,Y 520.227,Z 585.429,A -85,B 0,C 180,E1 5243.957,E2 5243.957} C_VEL
LIN {X 0,Y 520.281,Z 551.581,A -85,B 0,C 180,E1 5244.81,E2 5244.81} C_VEL
LIN {X 0,Y 513.747,Z 534.323,A -85,B 0,C 180,E1 5245.406,E2 5245.406} C_VEL
LIN {X 0,Y 510.338,Z 529.475,A -85,B 0,C 180,E1 5245.996,E2 5245.996} C_VEL
LIN {X 0,Y 507.355,Z 528.199,A -85,B 0,C 180,E1 5246.894,E2 5246.894} C_VEL
LIN {X 0,Y 504.349,Z 529.66,A -85,B 0,C 180,E1 5249.099,E2 5249.099} C_VEL
LIN {X 0,Y 504.331,Z 529.66,A -85,B 0,C 180,E1 5254.642,E2 5254.642} C_VEL
LIN {X 0,Y 504.17,Z 529.66,A -85,B 0,C 180,E1 5261.179,E2 5261.179} C_VEL
LIN {X 0,Y 504.227,Z 529.66,A -85,B 0,C 180,E1 5266.504,E2 5266.504} C_VEL
LIN {X 0,Y 504.377,Z 529.66,A -85,B 0,C 180,E1 5271.078,E2 5271.078} C_VEL
LIN {X 0,Y 504.29,Z 529.66,A -85,B 0,C 180,E1 5276.908,E2 5276.908} C_VEL
LIN {X 0,Y 504.467,Z 529.66,A -85,B 0,C 180,E1 5279.367,E2 5279.367} C_VEL
LIN {X 0,Y 514.619,Z 556.784,A -85,B 0,C 180,E1 5280.246,E2 5280.246} C_VEL
LIN {X 0,Y 516.223,Z 562.842,A -85,B 0,C 180,E1 5280.405,E2 5280.405} C_VEL
LIN {X 0,Y 515.403,Z 603.283,A -85,B 0,C 180,E1 5281.278,E2 5281.278} C_VEL
LIN {X 0,Y 513.942,Z 640.048,A -85,B 0,C 180,E1 5282.752,E2 5282.752} C_VEL
LIN {X 0,Y 512.056,Z 674.38,A -85,B 0,C 180,E1 5284.821,E2 5284.821} C_VEL
LIN {X 0,Y 509.907,Z 704.922,A -85,B 0,C 180,E1 5287.489,E2 5287.489} C_VEL
LIN {X 0,Y 507.972,Z 732.005,A -85,B 0,C 180,E1 5290.703,E2 5290.703} C_VEL
LIN {X 0,Y 506.475,Z 755.413,A -85,B 0,C 180,E1 5294.447,E2 5294.447} C_VEL
LIN {X 0,Y 505.597,Z 773.079,A -85,B 0,C 180,E1 5298.378,E2 5298.378} C_VEL
LIN {X 0,Y 505.295,Z 784.901,A -85,B 0,C 180,E1 5302.278,E2 5302.278} C_VEL
LIN {X 0,Y 505.195,Z 792.177,A -85,B 0,C 180,E1 5306.576,E2 5306.576} C_VEL
LIN {X 0,Y 505.094,Z 794,A -85,B 0,C 180,E1 5310.001,E2 5310.001} C_VEL
LIN {X 0,Y 505.197,Z 791.192,A -85,B 0,C 180,E1 5314.283,E2 5314.283} C_VEL
LIN {X 0,Y 505.353,Z 782.677,A -85,B 0,C 180,E1 5318.587,E2 5318.587} C_VEL
LIN {X 0,Y 505.747,Z 769.647,A -85,B 0,C 180,E1 5322.494,E2 5322.494} C_VEL
LIN {X 0,Y 506.695,Z 750.601,A -85,B 0,C 180,E1 5326.435,E2 5326.435} C_VEL
LIN {X 0,Y 508.226,Z 727.03,A -85,B 0,C 180,E1 5329.966,E2 5329.966} C_VEL
LIN {X 0,Y 510.314,Z 698.442,A -85,B 0,C 180,E1 5333.148,E2 5333.148} C_VEL
LIN {X 0,Y 512.406,Z 668.14,A -85,B 0,C 180,E1 5335.622,E2 5335.622} C_VEL
LIN {X 0,Y 514.46,Z 631.812,A -85,B 0,C 180,E1 5337.693,E2 5337.693} C_VEL
LIN {X 0,Y 515.927,Z 595.894,A -85,B 0,C 180,E1 5339.016,E2 5339.016} C_VEL
LIN {X 0,Y 516.151,Z 559.489,A -85,B 0,C 180,E1 5339.772,E2 5339.772} C_VEL
LIN {X 0,Y 504.427,Z 529.66,A -85,B 0,C 180,E1 5340.934,E2 5340.934} C_VEL
LIN {X 0,Y 504.417,Z 529.66,A -85,B 0,C 180,E1 5346.75,E2 5346.75} C_VEL
LIN {X 0,Y 504.247,Z 529.66,A -85,B 0,C 180,E1 5351.575,E2 5351.575} C_VEL
LIN {X 0,Y 504.232,Z 529.66,A -85,B 0,C 180,E1 5356.507,E2 5356.507} C_VEL
LIN {X 0,Y 504.386,Z 529.66,A -85,B 0,C 180,E1 5363.252,E2 5363.252} C_VEL
LIN {X 0,Y 504.351,Z 529.66,A -85,B 0,C 180,E1 5369.43,E2 5369.43} C_VEL
LIN {X 0,Y 504.432,Z 529.66,A -85,B 0,C 180,E1 5375.244,E2 5375.244} C_VEL
LIN {X 0,Y 504.659,Z 529.66,A -85,B 0,C 180,E1 5380.8,E2 5380.8} C_VEL
LIN {X 0,Y 504.474,Z 529.66,A -85,B 0,C 180,E1 5386.157,E2 5386.157} C_VEL
LIN {X 0,Y 504.702,Z 529.66,A -85,B 0,C 180,E1 5391.405,E2 5391.405} C_VEL
LIN {X 0,Y 504.859,Z 529.66,A -85,B 0,C 180,E1 5396.575,E2 5396.575} C_VEL
LIN {X 0,Y 504.883,Z 529.66,A -85,B 0,C 180,E1 5401.715,E2 5401.715} C_VEL
LIN {X 0,Y 504.782,Z 529.66,A -85,B 0,C 180,E1 5406.87,E2 5406.87} C_VEL
LIN {X 0,Y 504.719,Z 529.66,A -85,B 0,C 180,E1 5412.083,E2 5412.083} C_VEL
LIN {X 0,Y 504.679,Z 529.66,A -85,B 0,C 180,E1 5417.4,E2 5417.4} C_VEL
LIN {X 0,Y 504.506,Z 529.66,A -85,B 0,C 180,E1 5422.884,E2 5422.884} C_VEL
LIN {X 0,Y 504.333,Z 529.66,A -85,B 0,C 180,E1 5428.605,E2 5428.605} C_VEL
LIN {X 0,Y 504.303,Z 529.66,A -85,B 0,C 180,E1 5434.65,E2 5434.65} C_VEL
LIN {X 0,Y 504.165,Z 529.66,A -85,B 0,C 180,E1 5441.186,E2 5441.186} C_VEL
LIN {X 0,Y 504.542,Z 529.679,A -85,B 0,C 180,E1 5445.989,E2 5445.989} C_VEL
LIN {X 0,Y 509.75,Z 551.031,A -85,B 0,C 180,E1 5446.504,E2 5446.504} C_VEL
LIN {X 0,Y 509.416,Z 624.788,A -85,B 0,C 180,E1 5447.662,E2 5447.662} C_VEL
LIN {X 0,Y 508.628,Z 653.961,A -85,B 0,C 180,E1 5448.789,E2 5448.789} C_VEL
LIN {X 0,Y 507.65,Z 680.411,A -85,B 0,C 180,E1 5450.546,E2 5450.546} C_VEL
LIN {X 0,Y 506.638,Z 702.829,A -85,B 0,C 180,E1 5452.802,E2 5452.802} C_VEL
LIN {X 0,Y 505.937,Z 720.812,A -85,B 0,C 180,E1 5455.48,E2 5455.48} C_VEL
LIN {X 0,Y 505.545,Z 733.693,A -85,B 0,C 180,E1 5458.383,E2 5458.383} C_VEL
LIN {X 0,Y 505.263,Z 741.668,A -85,B 0,C 180,E1 5461.454,E2 5461.454} C_VEL
LIN {X 0,Y 505.081,Z 744.323,A -85,B 0,C 180,E1 5463.678,E2 5463.678} C_VEL
LIN {X 0,Y 505.073,Z 743.547,A -85,B 0,C 180,E1 5467.144,E2 5467.144} C_VEL
LIN {X 0,Y 505.376,Z 737.384,A -85,B 0,C 180,E1 5470.351,E2 5470.351} C_VEL
LIN {X 0,Y 505.743,Z 725.1,A -85,B 0,C 180,E1 5473.591,E2 5473.591} C_VEL
LIN {X 0,Y 506.408,Z 708.02,A -85,B 0,C 180,E1 5476.428,E2 5476.428} C_VEL
LIN {X 0,Y 507.338,Z 687.121,A -85,B 0,C 180,E1 5478.773,E2 5478.773} C_VEL
LIN {X 0,Y 508.367,Z 661.217,A -85,B 0,C 180,E1 5480.711,E2 5480.711} C_VEL
LIN {X 0,Y 509.248,Z 632.846,A -85,B 0,C 180,E1 5482.009,E2 5482.009} C_VEL
LIN {X 0,Y 509.617,Z 600.146,A -85,B 0,C 180,E1 5482.696,E2 5482.696} C_VEL
LIN {X 0,Y 508.924,Z 546.08,A -85,B 0,C 180,E1 5483.509,E2 5483.509} C_VEL
LIN {X 0,Y 504.589,Z 529.66,A -85,B 0,C 180,E1 5483.991,E2 5483.991} C_VEL
LIN {X 0,Y 504.846,Z 529.66,A -85,B 0,C 180,E1 5488.286,E2 5488.286} C_VEL
LIN {X 0,Y 504.88,Z 529.66,A -85,B 0,C 180,E1 5493.426,E2 5493.426} C_VEL
LIN {X 0,Y 504.691,Z 529.66,A -85,B 0,C 180,E1 5499.353,E2 5499.353} C_VEL
LIN {X 0,Y 504.573,Z 529.66,A -85,B 0,C 180,E1 5505.613,E2 5505.613} C_VEL
LIN {X 0,Y 504.54,Z 529.66,A -85,B 0,C 180,E1 5511.032,E2 5511.032} C_VEL
LIN {X 0,Y 504.36,Z 529.66,A -85,B 0,C 180,E1 5516.665,E2 5516.665} C_VEL
LIN {X 0,Y 504.266,Z 529.66,A -85,B 0,C 180,E1 5523.079,E2 5523.079} C_VEL
LIN {X 0,Y 504.385,Z 529.66,A -85,B 0,C 180,E1 5528.933,E2 5528.933} C_VEL
LIN {X 0,Y 504.265,Z 529.66,A -85,B 0,C 180,E1 5535.904,E2 5535.904} C_VEL
LIN {X 0,Y 504.333,Z 529.66,A -85,B 0,C 180,E1 5541.071,E2 5541.071} C_VEL
LIN {X 0,Y 504.236,Z 529.66,A -85,B 0,C 180,E1 5546.921,E2 5546.921} C_VEL
LIN {X 0,Y 504.467,Z 529.66,A -85,B 0,C 180,E1 5553.338,E2 5553.338} C_VEL
LIN {X 0,Y 504.548,Z 529.66,A -85,B 0,C 180,E1 5553.925,E2 5553.925} C_VEL
LIN {X 0,Y 513.878,Z 556.396,A -85,B 0,C 180,E1 5554.854,E2 5554.854} C_VEL
LIN {X 0,Y 512.799,Z 591.495,A -85,B 0,C 180,E1 5555.813,E2 5555.813} C_VEL
LIN {X 0,Y 511.232,Z 624.866,A -85,B 0,C 180,E1 5557.434,E2 5557.434} C_VEL
LIN {X 0,Y 509.353,Z 656.274,A -85,B 0,C 180,E1 5559.74,E2 5559.74} C_VEL
LIN {X 0,Y 507.699,Z 682.932,A -85,B 0,C 180,E1 5562.499,E2 5562.499} C_VEL
LIN {X 0,Y 506.436,Z 705.508,A -85,B 0,C 180,E1 5565.735,E2 5565.735} C_VEL
LIN {X 0,Y 505.642,Z 722.928,A -85,B 0,C 180,E1 5569.248,E2 5569.248} C_VEL
LIN {X 0,Y 505.369,Z 734.541,A -85,B 0,C 180,E1 5572.707,E2 5572.707} C_VEL
LIN {X 0,Y 505.224,Z 741.935,A -85,B 0,C 180,E1 5576.573,E2 5576.573} C_VEL
LIN {X 0,Y 505.115,Z 743.998,A -85,B 0,C 180,E1 5579.998,E2 5579.998} C_VEL
LIN {X 0,Y 505.228,Z 741.835,A -85,B 0,C 180,E1 5583.422,E2 5583.422} C_VEL
LIN {X 0,Y 505.392,Z 734.318,A -85,B 0,C 180,E1 5587.288,E2 5587.288} C_VEL
LIN {X 0,Y 505.824,Z 720.794,A -85,B 0,C 180,E1 5591.179,E2 5591.179} C_VEL
LIN {X 0,Y 506.679,Z 701.864,A -85,B 0,C 180,E1 5594.774,E2 5594.774} C_VEL
LIN {X 0,Y 507.975,Z 678.304,A -85,B 0,C 180,E1 5597.952,E2 5597.952} C_VEL
LIN {X 0,Y 509.746,Z 650.105,A -85,B 0,C 180,E1 5600.692,E2 5600.692} C_VEL
LIN {X 0,Y 511.484,Z 619.862,A -85,B 0,C 180,E1 5602.764,E2 5602.764} C_VEL
LIN {X 0,Y 513.012,Z 585.442,A -85,B 0,C 180,E1 5604.315,E2 5604.315} C_VEL
LIN {X 0,Y 513.319,Z 554.063,A -85,B 0,C 180,E1 5605.123,E2 5605.123} C_VEL
LIN {X 0,Y 504.476,Z 529.66,A -85,B 0,C 180,E1 5606.037,E2 5606.037} C_VEL
LIN {X 0,Y 504.349,Z 529.66,A -85,B 0,C 180,E1 5609.099,E2 5609.099} C_VEL
LIN {X 0,Y 501.777,Z 529.66,A -85,B 0,C 180,E1 5610.567,E2 5610.567} C_VEL
LIN {X 0,Y 496.472,Z 529.66,A -85,B 0,C 180,E1 5612.769,E2 5612.769} C_VEL
LIN {X 0,Y 496.406,Z 529.66,A -85,B 0,C 180,E1 5613.024,E2 5613.024} C_VEL
LIN {X 0,Y 496.22,Z 529.66,A -85,B 0,C 180,E1 5619.684,E2 5619.684} C_VEL
LIN {X 0,Y 496.323,Z 529.66,A -85,B 0,C 180,E1 5625.632,E2 5625.632} C_VEL
LIN {X 0,Y 496.424,Z 529.66,A -85,B 0,C 180,E1 5632.211,E2 5632.211} C_VEL
LIN {X 0,Y 496.546,Z 529.66,A -85,B 0,C 180,E1 5638.983,E2 5638.983} C_VEL
LIN {X 0,Y 507.46,Z 559.301,A -85,B 0,C 180,E1 5639.962,E2 5639.962} C_VEL
LIN {X 0,Y 508.863,Z 564.842,A -85,B 0,C 180,E1 5640.108,E2 5640.108} C_VEL
LIN {X 0,Y 508.018,Z 603.224,A -85,B 0,C 180,E1 5640.966,E2 5640.966} C_VEL
LIN {X 0,Y 506.472,Z 639.536,A -85,B 0,C 180,E1 5642.437,E2 5642.437} C_VEL
LIN {X 0,Y 504.41,Z 675.232,A -85,B 0,C 180,E1 5644.619,E2 5644.619} C_VEL
LIN {X 0,Y 502.252,Z 706.865,A -85,B 0,C 180,E1 5647.36,E2 5647.36} C_VEL
LIN {X 0,Y 500.317,Z 732.131,A -85,B 0,C 180,E1 5650.414,E2 5650.414} C_VEL
LIN {X 0,Y 498.712,Z 755.411,A -85,B 0,C 180,E1 5654.198,E2 5654.198} C_VEL
LIN {X 0,Y 497.772,Z 773.079,A -85,B 0,C 180,E1 5658.193,E2 5658.193} C_VEL
LIN {X 0,Y 497.411,Z 784.901,A -85,B 0,C 180,E1 5662.154,E2 5662.154} C_VEL
LIN {X 0,Y 497.317,Z 792.176,A -85,B 0,C 180,E1 5666.522,E2 5666.522} C_VEL
LIN {X 0,Y 497.221,Z 794,A -85,B 0,C 180,E1 5670.001,E2 5670.001} C_VEL
LIN {X 0,Y 497.297,Z 791.192,A -85,B 0,C 180,E1 5674.351,E2 5674.351} C_VEL
LIN {X 0,Y 497.465,Z 782.677,A -85,B 0,C 180,E1 5678.724,E2 5678.724} C_VEL
LIN {X 0,Y 497.93,Z 769.646,A -85,B 0,C 180,E1 5682.693,E2 5682.693} C_VEL
LIN {X 0,Y 498.973,Z 750.602,A -85,B 0,C 180,E1 5686.697,E2 5686.697} C_VEL
LIN {X 0,Y 500.7,Z 726.008,A -85,B 0,C 180,E1 5690.414,E2 5690.414} C_VEL
LIN {X 0,Y 502.701,Z 700.175,A -85,B 0,C 180,E1 5693.304,E2 5693.304} C_VEL
LIN {X 0,Y 504.919,Z 668.659,A -85,B 0,C 180,E1 5695.902,E2 5695.902} C_VEL
LIN {X 0,Y 507.121,Z 632.604,A -85,B 0,C 180,E1 5698.008,E2 5698.008} C_VEL
LIN {X 0,Y 508.776,Z 595.742,A -85,B 0,C 180,E1 5699.392,E2 5699.392} C_VEL
LIN {X 0,Y 509.02,Z 561.599,A -85,B 0,C 180,E1 5700.127,E2 5700.127} C_VEL
LIN {X 0,Y 496.507,Z 529.66,A -85,B 0,C 180,E1 5701.363,E2 5701.363} C_VEL
LIN {X 0,Y 496.439,Z 529.66,A -85,B 0,C 180,E1 5707.791,E2 5707.791} C_VEL
LIN {X 0,Y 496.316,Z 529.66,A -85,B 0,C 180,E1 5714.371,E2 5714.371} C_VEL
LIN {X 0,Y 496.382,Z 529.66,A -85,B 0,C 180,E1 5720.331,E2 5720.331} C_VEL
LIN {X 0,Y 496.37,Z 529.66,A -85,B 0,C 180,E1 5726.827,E2 5726.827} C_VEL
LIN {X 0,Y 496.472,Z 529.66,A -85,B 0,C 180,E1 5732.879,E2 5732.879} C_VEL
LIN {X 0,Y 496.654,Z 529.66,A -85,B 0,C 180,E1 5738.62,E2 5738.62} C_VEL
LIN {X 0,Y 496.664,Z 529.66,A -85,B 0,C 180,E1 5744.133,E2 5744.133} C_VEL
LIN {X 0,Y 496.771,Z 529.66,A -85,B 0,C 180,E1 5749.501,E2 5749.501} C_VEL
LIN {X 0,Y 496.993,Z 529.66,A -85,B 0,C 180,E1 5754.776,E2 5754.776} C_VEL
LIN {X 0,Y 497.064,Z 529.66,A -85,B 0,C 180,E1 5760.002,E2 5760.002} C_VEL
LIN {X 0,Y 496.99,Z 529.66,A -85,B 0,C 180,E1 5765.228,E2 5765.228} C_VEL
LIN {X 0,Y 496.813,Z 529.66,A -85,B 0,C 180,E1 5770.503,E2 5770.503} C_VEL
LIN {X 0,Y 496.756,Z 529.66,A -85,B 0,C 180,E1 5775.868,E2 5775.868} C_VEL
LIN {X 0,Y 496.648,Z 529.66,A -85,B 0,C 180,E1 5781.385,E2 5781.385} C_VEL
LIN {X 0,Y 496.413,Z 529.66,A -85,B 0,C 180,E1 5787.13,E2 5787.13} C_VEL
LIN {X 0,Y 496.387,Z 529.66,A -85,B 0,C 180,E1 5793.177,E2 5793.177} C_VEL
LIN {X 0,Y 496.196,Z 529.66,A -85,B 0,C 180,E1 5799.693,E2 5799.693} C_VEL
LIN {X 0,Y 496.58,Z 529.66,A -85,B 0,C 180,E1 5805.659,E2 5805.659} C_VEL
LIN {X 0,Y 502.385,Z 553.886,A -85,B 0,C 180,E1 5806.263,E2 5806.263} C_VEL
LIN {X 0,Y 501.855,Z 627.117,A -85,B 0,C 180,E1 5807.45,E2 5807.45} C_VEL
LIN {X 0,Y 501.009,Z 655.867,A -85,B 0,C 180,E1 5808.624,E2 5808.624} C_VEL
LIN {X 0,Y 500.003,Z 680.935,A -85,B 0,C 180,E1 5810.335,E2 5810.335} C_VEL
LIN {X 0,Y 498.943,Z 702.514,A -85,B 0,C 180,E1 5812.528,E2 5812.528} C_VEL
LIN {X 0,Y 498.155,Z 720.371,A -85,B 0,C 180,E1 5815.175,E2 5815.175} C_VEL
LIN {X 0,Y 497.685,Z 733.482,A -85,B 0,C 180,E1 5818.102,E2 5818.102} C_VEL
LIN {X 0,Y 497.431,Z 741.282,A -85,B 0,C 180,E1 5820.962,E2 5820.962} C_VEL
LIN {X 0,Y 497.23,Z 744.117,A -85,B 0,C 180,E1 5822.92,E2 5822.92} C_VEL
LIN {X 0,Y 497.091,Z 745.027,A -85,B 0,C 180,E1 5825.605,E2 5825.605} C_VEL
LIN {X 0,Y 497.375,Z 741.795,A -85,B 0,C 180,E1 5828.649,E2 5828.649} C_VEL
LIN {X 0,Y 497.647,Z 733.157,A -85,B 0,C 180,E1 5831.891,E2 5831.891} C_VEL
LIN {X 0,Y 498.237,Z 718.798,A -85,B 0,C 180,E1 5834.997,E2 5834.997} C_VEL
LIN {X 0,Y 499.107,Z 699.053,A -85,B 0,C 180,E1 5837.781,E2 5837.781} C_VEL
LIN {X 0,Y 500.228,Z 675.4,A -85,B 0,C 180,E1 5840.011,E2 5840.011} C_VEL
LIN {X 0,Y 501.22,Z 648.204,A -85,B 0,C 180,E1 5841.669,E2 5841.669} C_VEL
LIN {X 0,Y 501.971,Z 619.049,A -85,B 0,C 180,E1 5842.66,E2 5842.66} C_VEL
LIN {X 0,Y 501.492,Z 547.587,A -85,B 0,C 180,E1 5843.773,E2 5843.773} C_VEL
LIN {X 0,Y 496.728,Z 529.66,A -85,B 0,C 180,E1 5844.279,E2 5844.279} C_VEL
LIN {X 0,Y 497.069,Z 529.66,A -85,B 0,C 180,E1 5849.999,E2 5849.999} C_VEL
LIN {X 0,Y 497.037,Z 529.66,A -85,B 0,C 180,E1 5855.225,E2 5855.225} C_VEL
LIN {X 0,Y 496.799,Z 529.66,A -85,B 0,C 180,E1 5860.5,E2 5860.5} C_VEL
LIN {X 0,Y 496.674,Z 529.66,A -85,B 0,C 180,E1 5865.868,E2 5865.868} C_VEL
LIN {X 0,Y 496.624,Z 529.66,A -85,B 0,C 180,E1 5871.383,E2 5871.383} C_VEL
LIN {X 0,Y 496.394,Z 529.66,A -85,B 0,C 180,E1 5877.128,E2 5877.128} C_VEL
LIN {X 0,Y 496.36,Z 529.66,A -85,B 0,C 180,E1 5883.176,E2 5883.176} C_VEL
LIN {X 0,Y 496.388,Z 529.66,A -85,B 0,C 180,E1 5889.671,E2 5889.671} C_VEL
LIN {X 0,Y 496.349,Z 529.66,A -85,B 0,C 180,E1 5895.631,E2 5895.631} C_VEL
LIN {X 0,Y 496.334,Z 529.66,A -85,B 0,C 180,E1 5900.321,E2 5900.321} C_VEL
LIN {X 0,Y 496.327,Z 529.66,A -85,B 0,C 180,E1 5906.819,E2 5906.819} C_VEL
LIN {X 0,Y 496.595,Z 529.66,A -85,B 0,C 180,E1 5913.475,E2 5913.475} C_VEL
LIN {X 0,Y 506.613,Z 558.991,A -85,B 0,C 180,E1 5914.536,E2 5914.536} C_VEL
LIN {X 0,Y 505.438,Z 594.242,A -85,B 0,C 180,E1 5915.566,E2 5915.566} C_VEL
LIN {X 0,Y 503.778,Z 626.631,A -85,B 0,C 180,E1 5917.202,E2 5917.202} C_VEL
LIN {X 0,Y 501.762,Z 657.496,A -85,B 0,C 180,E1 5919.534,E2 5919.534} C_VEL
LIN {X 0,Y 499.933,Z 684.544,A -85,B 0,C 180,E1 5922.43,E2 5922.43} C_VEL
LIN {X 0,Y 498.598,Z 706.699,A -85,B 0,C 180,E1 5925.719,E2 5925.719} C_VEL
LIN {X 0,Y 497.795,Z 722.923,A -85,B 0,C 180,E1 5929.077,E2 5929.077} C_VEL
LIN {X 0,Y 497.441,Z 735.631,A -85,B 0,C 180,E1 5933.028,E2 5933.028} C_VEL
LIN {X 0,Y 497.346,Z 741.931,A -85,B 0,C 180,E1 5936.519,E2 5936.519} C_VEL
LIN {X 0,Y 497.241,Z 743.998,A -85,B 0,C 180,E1 5939.998,E2 5939.998} C_VEL
LIN {X 0,Y 497.351,Z 741.833,A -85,B 0,C 180,E1 5943.477,E2 5943.477} C_VEL
LIN {X 0,Y 497.506,Z 734.317,A -85,B 0,C 180,E1 5947.404,E2 5947.404} C_VEL
LIN {X 0,Y 497.969,Z 720.799,A -85,B 0,C 180,E1 5951.357,E2 5951.357} C_VEL
LIN {X 0,Y 498.962,Z 701.506,A -85,B 0,C 180,E1 5955.065,E2 5955.065} C_VEL
LIN {X 0,Y 500.37,Z 678.307,A -85,B 0,C 180,E1 5958.234,E2 5958.234} C_VEL
LIN {X 0,Y 502.253,Z 650.112,A -85,B 0,C 180,E1 5961.015,E2 5961.015} C_VEL
LIN {X 0,Y 504.106,Z 620.254,A -85,B 0,C 180,E1 5963.086,E2 5963.086} C_VEL
LIN {X 0,Y 505.681,Z 586.526,A -85,B 0,C 180,E1 5964.622,E2 5964.622} C_VEL
LIN {X 0,Y 505.933,Z 555.643,A -85,B 0,C 180,E1 5965.45,E2 5965.45} C_VEL
LIN {X 0,Y 496.532,Z 529.66,A -85,B 0,C 180,E1 5966.396,E2 5966.396} C_VEL
LIN {X 0,Y 496.406,Z 529.66,A -85,B 0,C 180,E1 5973.024,E2 5973.024} C_VEL
LIN {X 0,Y 493.928,Z 529.66,A -85,B 0,C 180,E1 5974.503,E2 5974.503} C_VEL
LIN {X 0,Y 488.424,Z 529.66,A -85,B 0,C 180,E1 5976.721,E2 5976.721} C_VEL
LIN {X 0,Y 488.311,Z 529.66,A -85,B 0,C 180,E1 5976.978,E2 5976.978} C_VEL
LIN {X 0,Y 488.332,Z 529.66,A -85,B 0,C 180,E1 5982.826,E2 5982.826} C_VEL
LIN {X 0,Y 488.418,Z 529.66,A -85,B 0,C 180,E1 5987.854,E2 5987.854} C_VEL
LIN {X 0,Y 488.445,Z 529.66,A -85,B 0,C 180,E1 5994.058,E2 5994.058} C_VEL
LIN {X 0,Y 488.63,Z 529.66,A -85,B 0,C 180,E1 5998.57,E2 5998.57} C_VEL
LIN {X 0,Y 500.643,Z 562.509,A -85,B 0,C 180,E1 5999.696,E2 5999.696} C_VEL
LIN {X 0,Y 501.33,Z 579.733,A -85,B 0,C 180,E1 6000.035,E2 6000.035} C_VEL
LIN {X 0,Y 500.073,Z 617.037,A -85,B 0,C 180,E1 6001.132,E2 6001.132} C_VEL
LIN {X 0,Y 498.252,Z 652.707,A -85,B 0,C 180,E1 6002.86,E2 6002.86} C_VEL
LIN {X 0,Y 495.978,Z 687.381,A -85,B 0,C 180,E1 6005.32,E2 6005.32} C_VEL
LIN {X 0,Y 493.766,Z 717.145,A -85,B 0,C 180,E1 6008.251,E2 6008.251} C_VEL
LIN {X 0,Y 491.992,Z 741.141,A -85,B 0,C 180,E1 6011.447,E2 6011.447} C_VEL
LIN {X 0,Y 490.509,Z 762.793,A -85,B 0,C 180,E1 6015.463,E2 6015.463} C_VEL
LIN {X 0,Y 489.755,Z 777.609,A -85,B 0,C 180,E1 6019.347,E2 6019.347} C_VEL
LIN {X 0,Y 489.478,Z 786.819,A -85,B 0,C 180,E1 6022.917,E2 6022.917} C_VEL
LIN {X 0,Y 489.412,Z 792.175,A -85,B 0,C 180,E1 6026.465,E2 6026.465} C_VEL
LIN {X 0,Y 489.321,Z 794,A -85,B 0,C 180,E1 6030.001,E2 6030.001} C_VEL
LIN {X 0,Y 489.396,Z 791.192,A -85,B 0,C 180,E1 6034.422,E2 6034.422} C_VEL
LIN {X 0,Y 489.583,Z 782.677,A -85,B 0,C 180,E1 6038.866,E2 6038.866} C_VEL
LIN {X 0,Y 490.102,Z 769.646,A -85,B 0,C 180,E1 6042.899,E2 6042.899} C_VEL
LIN {X 0,Y 491.264,Z 750.602,A -85,B 0,C 180,E1 6046.967,E2 6046.967} C_VEL
LIN {X 0,Y 492.923,Z 728.025,A -85,B 0,C 180,E1 6050.44,E2 6050.44} C_VEL
LIN {X 0,Y 495.193,Z 699.274,A -85,B 0,C 180,E1 6053.674,E2 6053.674} C_VEL
LIN {X 0,Y 497.667,Z 666.572,A -85,B 0,C 180,E1 6056.378,E2 6056.378} C_VEL
LIN {X 0,Y 499.96,Z 630.924,A -85,B 0,C 180,E1 6058.446,E2 6058.446} C_VEL
LIN {X 0,Y 501.667,Z 594.994,A -85,B 0,C 180,E1 6059.796,E2 6059.796} C_VEL
LIN {X 0,Y 501.927,Z 563.76,A -85,B 0,C 180,E1 6060.49,E2 6060.49} C_VEL
LIN {X 0,Y 488.525,Z 529.66,A -85,B 0,C 180,E1 6061.945,E2 6061.945} C_VEL
LIN {X 0,Y 488.507,Z 529.66,A -85,B 0,C 180,E1 6068.156,E2 6068.156} C_VEL
LIN {X 0,Y 488.405,Z 529.66,A -85,B 0,C 180,E1 6074.719,E2 6074.719} C_VEL
LIN {X 0,Y 488.458,Z 529.66,A -85,B 0,C 180,E1 6080.564,E2 6080.564} C_VEL
LIN {X 0,Y 488.462,Z 529.66,A -85,B 0,C 180,E1 6086.524,E2 6086.524} C_VEL
LIN {X 0,Y 488.542,Z 529.66,A -85,B 0,C 180,E1 6092.402,E2 6092.402} C_VEL
LIN {X 0,Y 488.689,Z 529.66,A -85,B 0,C 180,E1 6098.254,E2 6098.254} C_VEL
LIN {X 0,Y 488.747,Z 529.66,A -85,B 0,C 180,E1 6103.869,E2 6103.869} C_VEL
LIN {X 0,Y 488.848,Z 529.66,A -85,B 0,C 180,E1 6109.329,E2 6109.329} C_VEL
LIN {X 0,Y 489.081,Z 529.66,A -85,B 0,C 180,E1 6114.691,E2 6114.691} C_VEL
LIN {X 0,Y 489.164,Z 529.66,A -85,B 0,C 180,E1 6120.002,E2 6120.002} C_VEL
LIN {X 0,Y 489.075,Z 529.66,A -85,B 0,C 180,E1 6125.313,E2 6125.313} C_VEL
LIN {X 0,Y 488.897,Z 529.66,A -85,B 0,C 180,E1 6130.675,E2 6130.675} C_VEL
LIN {X 0,Y 488.787,Z 529.66,A -85,B 0,C 180,E1 6136.853,E2 6136.853} C_VEL
LIN {X 0,Y 488.672,Z 529.66,A -85,B 0,C 180,E1 6142.12,E2 6142.12} C_VEL
LIN {X 0,Y 488.492,Z 529.66,A -85,B 0,C 180,E1 6147.607,E2 6147.607} C_VEL
LIN {X 0,Y 488.457,Z 529.66,A -85,B 0,C 180,E1 6153.787,E2 6153.787} C_VEL
LIN {X 0,Y 488.313,Z 529.66,A -85,B 0,C 180,E1 6160.465,E2 6160.465} C_VEL
LIN {X 0,Y 488.634,Z 529.929,A -85,B 0,C 180,E1 6165.345,E2 6165.345} C_VEL
LIN {X 0,Y 494.809,Z 552.425,A -85,B 0,C 180,E1 6165.942,E2 6165.942} C_VEL
LIN {X 0,Y 494.349,Z 626.685,A -85,B 0,C 180,E1 6167.156,E2 6167.156} C_VEL
LIN {X 0,Y 493.446,Z 655.784,A -85,B 0,C 180,E1 6168.344,E2 6168.344} C_VEL
LIN {X 0,Y 492.308,Z 682.386,A -85,B 0,C 180,E1 6170.195,E2 6170.195} C_VEL
LIN {X 0,Y 491.111,Z 705.162,A -85,B 0,C 180,E1 6172.623,E2 6172.623} C_VEL
LIN {X 0,Y 490.226,Z 723.515,A -85,B 0,C 180,E1 6175.546,E2 6175.546} C_VEL
LIN {X 0,Y 489.785,Z 735.279,A -85,B 0,C 180,E1 6178.414,E2 6178.414} C_VEL
LIN {X 0,Y 489.527,Z 742.078,A -85,B 0,C 180,E1 6181.127,E2 6181.127} C_VEL
LIN {X 0,Y 489.211,Z 745.437,A -85,B 0,C 180,E1 6184.415,E2 6184.415} C_VEL
LIN {X 0,Y 489.346,Z 743.74,A -85,B 0,C 180,E1 6187.689,E2 6187.689} C_VEL
LIN {X 0,Y 489.714,Z 736.4,A -85,B 0,C 180,E1 6191.122,E2 6191.122} C_VEL
LIN {X 0,Y 490.246,Z 723.374,A -85,B 0,C 180,E1 6194.375,E2 6194.375} C_VEL
LIN {X 0,Y 491.135,Z 704.543,A -85,B 0,C 180,E1 6197.354,E2 6197.354} C_VEL
LIN {X 0,Y 492.289,Z 682.006,A -85,B 0,C 180,E1 6199.736,E2 6199.736} C_VEL
LIN {X 0,Y 493.49,Z 655.146,A -85,B 0,C 180,E1 6201.592,E2 6201.592} C_VEL
LIN {X 0,Y 494.34,Z 626.145,A -85,B 0,C 180,E1 6202.766,E2 6202.766} C_VEL
LIN {X 0,Y 493.972,Z 548.778,A -85,B 0,C 180,E1 6204.055,E2 6204.055} C_VEL
LIN {X 0,Y 488.848,Z 529.66,A -85,B 0,C 180,E1 6204.56,E2 6204.56} C_VEL
LIN {X 0,Y 489.168,Z 529.66,A -85,B 0,C 180,E1 6209.999,E2 6209.999} C_VEL
LIN {X 0,Y 489.123,Z 529.66,A -85,B 0,C 180,E1 6215.31,E2 6215.31} C_VEL
LIN {X 0,Y 488.88,Z 529.66,A -85,B 0,C 180,E1 6220.672,E2 6220.672} C_VEL
LIN {X 0,Y 488.724,Z 529.66,A -85,B 0,C 180,E1 6226.826,E2 6226.826} C_VEL
LIN {X 0,Y 488.652,Z 529.66,A -85,B 0,C 180,E1 6232.112,E2 6232.112} C_VEL
LIN {X 0,Y 488.47,Z 529.66,A -85,B 0,C 180,E1 6237.605,E2 6237.605} C_VEL
LIN {X 0,Y 488.455,Z 529.66,A -85,B 0,C 180,E1 6243.784,E2 6243.784} C_VEL
LIN {X 0,Y 488.467,Z 529.66,A -85,B 0,C 180,E1 6249.435,E2 6249.435} C_VEL
LIN {X 0,Y 488.428,Z 529.66,A -85,B 0,C 180,E1 6255.281,E2 6255.281} C_VEL
LIN {X 0,Y 488.407,Z 529.66,A -85,B 0,C 180,E1 6261.833,E2 6261.833} C_VEL
LIN {X 0,Y 488.401,Z 529.66,A -85,B 0,C 180,E1 6268.313,E2 6268.313} C_VEL
LIN {X 0,Y 488.612,Z 529.66,A -85,B 0,C 180,E1 6273.04,E2 6273.04} C_VEL
LIN {X 0,Y 499.408,Z 560.147,A -85,B 0,C 180,E1 6274.188,E2 6274.188} C_VEL
LIN {X 0,Y 498.13,Z 595.205,A -85,B 0,C 180,E1 6275.247,E2 6275.247} C_VEL
LIN {X 0,Y 496.305,Z 628.054,A -85,B 0,C 180,E1 6276.953,E2 6276.953} C_VEL
LIN {X 0,Y 494.183,Z 658.68,A -85,B 0,C 180,E1 6279.323,E2 6279.323} C_VEL
LIN {X 0,Y 492.3,Z 684.535,A -85,B 0,C 180,E1 6282.148,E2 6282.148} C_VEL
LIN {X 0,Y 490.813,Z 706.958,A -85,B 0,C 180,E1 6285.536,E2 6285.536} C_VEL
LIN {X 0,Y 489.973,Z 722.918,A -85,B 0,C 180,E1 6288.9,E2 6288.9} C_VEL
LIN {X 0,Y 489.579,Z 734.816,A -85,B 0,C 180,E1 6292.586,E2 6292.586} C_VEL
LIN {X 0,Y 489.442,Z 741.927,A -85,B 0,C 180,E1 6296.462,E2 6296.462} C_VEL
LIN {X 0,Y 489.341,Z 743.998,A -85,B 0,C 180,E1 6299.998,E2 6299.998} C_VEL
LIN {X 0,Y 489.448,Z 741.83,A -85,B 0,C 180,E1 6303.533,E2 6303.533} C_VEL
LIN {X 0,Y 489.621,Z 734.316,A -85,B 0,C 180,E1 6307.524,E2 6307.524} C_VEL
LIN {X 0,Y 490.121,Z 720.803,A -85,B 0,C 180,E1 6311.542,E2 6311.542} C_VEL
LIN {X 0,Y 491.198,Z 701.972,A -85,B 0,C 180,E1 6315.233,E2 6315.233} C_VEL
LIN {X 0,Y 492.752,Z 678.789,A -85,B 0,C 180,E1 6318.469,E2 6318.469} C_VEL
LIN {X 0,Y 494.687,Z 651.341,A -85,B 0,C 180,E1 6321.235,E2 6321.235} C_VEL
LIN {X 0,Y 496.754,Z 619.951,A -85,B 0,C 180,E1 6323.435,E2 6323.435} C_VEL
LIN {X 0,Y 498.4,Z 585.885,A -85,B 0,C 180,E1 6324.99,E2 6324.99} C_VEL
LIN {X 0,Y 498.704,Z 557.813,A -85,B 0,C 180,E1 6325.764,E2 6325.764} C_VEL
LIN {X 0,Y 488.605,Z 529.66,A -85,B 0,C 180,E1 6326.816,E2 6326.816} C_VEL
LIN {X 0,Y 488.497,Z 529.66,A -85,B 0,C 180,E1 6333.485,E2 6333.485} C_VEL
LIN {X 0,Y 488.311,Z 529.66,A -85,B 0,C 180,E1 6336.978,E2 6336.978} C_VEL
LIN {X 0,Y 486.987,Z 529.66,A -85,B 0,C 180,E1 6337.991,E2 6337.991} C_VEL
LIN {X 0,Y 480.443,Z 529.66,A -85,B 0,C 180,E1 6340.754,E2 6340.754} C_VEL
LIN {X 0,Y 480.386,Z 529.66,A -85,B 0,C 180,E1 6341.016,E2 6341.016} C_VEL
LIN {X 0,Y 480.453,Z 529.66,A -85,B 0,C 180,E1 6346.294,E2 6346.294} C_VEL
LIN {X 0,Y 480.601,Z 529.66,A -85,B 0,C 180,E1 6351.711,E2 6351.711} C_VEL
LIN {X 0,Y 480.672,Z 529.66,A -85,B 0,C 180,E1 6358.127,E2 6358.127} C_VEL
LIN {X 0,Y 494.201,Z 568.005,A -85,B 0,C 180,E1 6359.481,E2 6359.481} C_VEL
LIN {X 0,Y 493.135,Z 606.564,A -85,B 0,C 180,E1 6360.428,E2 6360.428} C_VEL
LIN {X 0,Y 491.34,Z 643.311,A -85,B 0,C 180,E1 6362.027,E2 6362.027} C_VEL
LIN {X 0,Y 489.068,Z 677.483,A -85,B 0,C 180,E1 6364.257,E2 6364.257} C_VEL
LIN {X 0,Y 486.745,Z 708.509,A -85,B 0,C 180,E1 6367.08,E2 6367.08} C_VEL
LIN {X 0,Y 484.689,Z 735.767,A -85,B 0,C 180,E1 6370.448,E2 6370.448} C_VEL
LIN {X 0,Y 483.042,Z 757.672,A -85,B 0,C 180,E1 6374.137,E2 6374.137} C_VEL
LIN {X 0,Y 482.017,Z 774.608,A -85,B 0,C 180,E1 6378.26,E2 6378.26} C_VEL
LIN {X 0,Y 481.665,Z 784.901,A -85,B 0,C 180,E1 6381.896,E2 6381.896} C_VEL
LIN {X 0,Y 481.533,Z 792.175,A -85,B 0,C 180,E1 6386.407,E2 6386.407} C_VEL
LIN {X 0,Y 481.427,Z 794,A -85,B 0,C 180,E1 6390.001,E2 6390.001} C_VEL
LIN {X 0,Y 481.519,Z 791.191,A -85,B 0,C 180,E1 6394.494,E2 6394.494} C_VEL
LIN {X 0,Y 481.714,Z 782.677,A -85,B 0,C 180,E1 6399.012,E2 6399.012} C_VEL
LIN {X 0,Y 482.35,Z 768.353,A -85,B 0,C 180,E1 6403.454,E2 6403.454} C_VEL
LIN {X 0,Y 483.617,Z 749.292,A -85,B 0,C 180,E1 6407.426,E2 6407.426} C_VEL
LIN {X 0,Y 485.466,Z 724.912,A -85,B 0,C 180,E1 6411.076,E2 6411.076} C_VEL
LIN {X 0,Y 487.894,Z 696.527,A -85,B 0,C 180,E1 6414.234,E2 6414.234} C_VEL
LIN {X 0,Y 490.483,Z 663.544,A -85,B 0,C 180,E1 6416.926,E2 6416.926} C_VEL
LIN {X 0,Y 492.894,Z 628.003,A -85,B 0,C 180,E1 6418.954,E2 6418.954} C_VEL
LIN {X 0,Y 494.769,Z 590.849,A -85,B 0,C 180,E1 6420.306,E2 6420.306} C_VEL
LIN {X 0,Y 494.692,Z 565.511,A -85,B 0,C 180,E1 6420.88,E2 6420.88} C_VEL
LIN {X 0,Y 480.592,Z 529.66,A -85,B 0,C 180,E1 6422.416,E2 6422.416} C_VEL
LIN {X 0,Y 480.574,Z 529.66,A -85,B 0,C 180,E1 6428.903,E2 6428.903} C_VEL
LIN {X 0,Y 480.438,Z 529.66,A -85,B 0,C 180,E1 6433.751,E2 6433.751} C_VEL
LIN {X 0,Y 480.503,Z 529.66,A -85,B 0,C 180,E1 6438.914,E2 6438.914} C_VEL
LIN {X 0,Y 480.493,Z 529.66,A -85,B 0,C 180,E1 6444.74,E2 6444.74} C_VEL
LIN {X 0,Y 480.536,Z 529.66,A -85,B 0,C 180,E1 6449.842,E2 6449.842} C_VEL
LIN {X 0,Y 480.676,Z 529.66,A -85,B 0,C 180,E1 6455.917,E2 6455.917} C_VEL
LIN {X 0,Y 480.888,Z 529.66,A -85,B 0,C 180,E1 6461.715,E2 6461.715} C_VEL
LIN {X 0,Y 480.797,Z 529.66,A -85,B 0,C 180,E1 6467.311,E2 6467.311} C_VEL
LIN {X 0,Y 481.123,Z 529.66,A -85,B 0,C 180,E1 6472.795,E2 6472.795} C_VEL
LIN {X 0,Y 481.422,Z 529.66,A -85,B 0,C 180,E1 6478.206,E2 6478.206} C_VEL
LIN {X 0,Y 481.303,Z 529.66,A -85,B 0,C 180,E1 6483.597,E2 6483.597} C_VEL
LIN {X 0,Y 481.072,Z 529.66,A -85,B 0,C 180,E1 6489.026,E2 6489.026} C_VEL
LIN {X 0,Y 480.98,Z 529.66,A -85,B 0,C 180,E1 6494.538,E2 6494.538} C_VEL
LIN {X 0,Y 480.823,Z 529.66,A -85,B 0,C 180,E1 6500.197,E2 6500.197} C_VEL
LIN {X 0,Y 480.622,Z 529.66,A -85,B 0,C 180,E1 6506.078,E2 6506.078} C_VEL
LIN {X 0,Y 480.522,Z 529.66,A -85,B 0,C 180,E1 6512.269,E2 6512.269} C_VEL
LIN {X 0,Y 480.356,Z 529.66,A -85,B 0,C 180,E1 6518.926,E2 6518.926} C_VEL
LIN {X 0,Y 480.691,Z 529.66,A -85,B 0,C 180,E1 6524.976,E2 6524.976} C_VEL
LIN {X 0,Y 487.427,Z 555.144,A -85,B 0,C 180,E1 6525.682,E2 6525.682} C_VEL
LIN {X 0,Y 486.843,Z 627.671,A -85,B 0,C 180,E1 6526.893,E2 6526.893} C_VEL
LIN {X 0,Y 485.887,Z 656.366,A -85,B 0,C 180,E1 6528.092,E2 6528.092} C_VEL
LIN {X 0,Y 484.652,Z 682.724,A -85,B 0,C 180,E1 6529.955,E2 6529.955} C_VEL
LIN {X 0,Y 483.402,Z 705.185,A -85,B 0,C 180,E1 6532.376,E2 6532.376} C_VEL
LIN {X 0,Y 482.41,Z 723.882,A -85,B 0,C 180,E1 6535.389,E2 6535.389} C_VEL
LIN {X 0,Y 481.915,Z 736.21,A -85,B 0,C 180,E1 6538.474,E2 6538.474} C_VEL
LIN {X 0,Y 481.532,Z 743.867,A -85,B 0,C 180,E1 6541.961,E2 6541.961} C_VEL
LIN {X 0,Y 481.264,Z 745.839,A -85,B 0,C 180,E1 6545.411,E2 6545.411} C_VEL
LIN {X 0,Y 481.616,Z 742.368,A -85,B 0,C 180,E1 6548.88,E2 6548.88} C_VEL
LIN {X 0,Y 482.036,Z 732.753,A -85,B 0,C 180,E1 6552.432,E2 6552.432} C_VEL
LIN {X 0,Y 482.683,Z 718.436,A -85,B 0,C 180,E1 6555.516,E2 6555.516} C_VEL
LIN {X 0,Y 483.732,Z 698.89,A -85,B 0,C 180,E1 6558.3,E2 6558.3} C_VEL
LIN {X 0,Y 485.081,Z 674.669,A -85,B 0,C 180,E1 6560.6,E2 6560.6} C_VEL
LIN {X 0,Y 486.163,Z 647.797,A -85,B 0,C 180,E1 6562.252,E2 6562.252} C_VEL
LIN {X 0,Y 486.984,Z 618.973,A -85,B 0,C 180,E1 6563.231,E2 6563.231} C_VEL
LIN {X 0,Y 486.6,Z 550.534,A -85,B 0,C 180,E1 6564.329,E2 6564.329} C_VEL
LIN {X 0,Y 480.97,Z 529.66,A -85,B 0,C 180,E1 6564.937,E2 6564.937} C_VEL
LIN {X 0,Y 481.274,Z 529.66,A -85,B 0,C 180,E1 6569.999,E2 6569.999} C_VEL
LIN {X 0,Y 481.209,Z 529.66,A -85,B 0,C 180,E1 6575.397,E2 6575.397} C_VEL
LIN {X 0,Y 480.955,Z 529.66,A -85,B 0,C 180,E1 6580.85,E2 6580.85} C_VEL
LIN {X 0,Y 480.845,Z 529.66,A -85,B 0,C 180,E1 6586.405,E2 6586.405} C_VEL
LIN {X 0,Y 480.761,Z 529.66,A -85,B 0,C 180,E1 6592.126,E2 6592.126} C_VEL
LIN {X 0,Y 480.479,Z 529.66,A -85,B 0,C 180,E1 6598.43,E2 6598.43} C_VEL
LIN {X 0,Y 480.486,Z 529.66,A -85,B 0,C 180,E1 6604.422,E2 6604.422} C_VEL
LIN {X 0,Y 480.578,Z 529.66,A -85,B 0,C 180,E1 6608.901,E2 6608.901} C_VEL
LIN {X 0,Y 480.458,Z 529.66,A -85,B 0,C 180,E1 6613.747,E2 6613.747} C_VEL
LIN {X 0,Y 480.482,Z 529.66,A -85,B 0,C 180,E1 6618.914,E2 6618.914} C_VEL
LIN {X 0,Y 480.43,Z 529.66,A -85,B 0,C 180,E1 6624.748,E2 6624.748} C_VEL
LIN {X 0,Y 480.511,Z 529.66,A -85,B 0,C 180,E1 6629.835,E2 6629.835} C_VEL
LIN {X 0,Y 480.697,Z 529.66,A -85,B 0,C 180,E1 6632.592,E2 6632.592} C_VEL
LIN {X 0,Y 492.144,Z 562.7,A -85,B 0,C 180,E1 6633.859,E2 6633.859} C_VEL
LIN {X 0,Y 490.749,Z 597.821,A -85,B 0,C 180,E1 6634.988,E2 6634.988} C_VEL
LIN {X 0,Y 488.858,Z 629.546,A -85,B 0,C 180,E1 6636.701,E2 6636.701} C_VEL
LIN {X 0,Y 486.597,Z 660.21,A -85,B 0,C 180,E1 6639.143,E2 6639.143} C_VEL
LIN {X 0,Y 484.545,Z 686.293,A -85,B 0,C 180,E1 6642.087,E2 6642.087} C_VEL
LIN {X 0,Y 482.999,Z 708.19,A -85,B 0,C 180,E1 6645.524,E2 6645.524} C_VEL
LIN {X 0,Y 482.032,Z 724.671,A -85,B 0,C 180,E1 6649.172,E2 6649.172} C_VEL
LIN {X 0,Y 481.671,Z 735.622,A -85,B 0,C 180,E1 6652.799,E2 6652.799} C_VEL
LIN {X 0,Y 481.562,Z 741.922,A -85,B 0,C 180,E1 6656.405,E2 6656.405} C_VEL
LIN {X 0,Y 481.447,Z 743.998,A -85,B 0,C 180,E1 6659.998,E2 6659.998} C_VEL
LIN {X 0,Y 481.569,Z 741.828,A -85,B 0,C 180,E1 6663.591,E2 6663.591} C_VEL
LIN {X 0,Y 481.749,Z 734.315,A -85,B 0,C 180,E1 6667.648,E2 6667.648} C_VEL
LIN {X 0,Y 482.306,Z 720.806,A -85,B 0,C 180,E1 6671.731,E2 6671.731} C_VEL
LIN {X 0,Y 483.505,Z 701.238,A -85,B 0,C 180,E1 6675.613,E2 6675.613} C_VEL
LIN {X 0,Y 485.175,Z 678.475,A -85,B 0,C 180,E1 6678.808,E2 6678.808} C_VEL
LIN {X 0,Y 487.212,Z 651.373,A -85,B 0,C 180,E1 6681.556,E2 6681.556} C_VEL
LIN {X 0,Y 489.392,Z 619.864,A -85,B 0,C 180,E1 6683.782,E2 6683.782} C_VEL
LIN {X 0,Y 491.116,Z 585.935,A -85,B 0,C 180,E1 6685.343,E2 6685.343} C_VEL
LIN {X 0,Y 491.247,Z 559.303,A -85,B 0,C 180,E1 6686.112,E2 6686.112} C_VEL
LIN {X 0,Y 480.678,Z 529.66,A -85,B 0,C 180,E1 6687.272,E2 6687.272} C_VEL
LIN {X 0,Y 480.544,Z 529.66,A -85,B 0,C 180,E1 6692.261,E2 6692.261} C_VEL
LIN {X 0,Y 480.396,Z 529.66,A -85,B 0,C 180,E1 6698.916,E2 6698.916} C_VEL
LIN {X 0,Y 480.386,Z 529.66,A -85,B 0,C 180,E1 6701.016,E2 6701.016} C_VEL
LIN {X 0,Y 477.939,Z 529.66,A -85,B 0,C 180,E1 6702.549,E2 6702.549} C_VEL
LIN {X 0,Y 472.526,Z 529.66,A -85,B 0,C 180,E1 6704.85,E2 6704.85} C_VEL
LIN {X 0,Y 472.44,Z 529.66,A -85,B 0,C 180,E1 6705.116,E2 6705.116} C_VEL
LIN {X 0,Y 472.567,Z 529.66,A -85,B 0,C 180,E1 6710.311,E2 6710.311} C_VEL
LIN {X 0,Y 472.571,Z 529.66,A -85,B 0,C 180,E1 6716.116,E2 6716.116} C_VEL
LIN {X 0,Y 472.698,Z 529.66,A -85,B 0,C 180,E1 6717.661,E2 6717.661} C_VEL
LIN {X 0,Y 486.903,Z 570.058,A -85,B 0,C 180,E1 6719.162,E2 6719.162} C_VEL
LIN {X 0,Y 485.717,Z 607.591,A -85,B 0,C 180,E1 6720.126,E2 6720.126} C_VEL
LIN {X 0,Y 483.82,Z 644.822,A -85,B 0,C 180,E1 6721.8,E2 6721.8} C_VEL
LIN {X 0,Y 481.385,Z 678.933,A -85,B 0,C 180,E1 6724.095,E2 6724.095} C_VEL
LIN {X 0,Y 478.908,Z 710.418,A -85,B 0,C 180,E1 6727.051,E2 6727.051} C_VEL
LIN {X 0,Y 476.738,Z 737.864,A -85,B 0,C 180,E1 6730.589,E2 6730.589} C_VEL
LIN {X 0,Y 475.017,Z 760.291,A -85,B 0,C 180,E1 6734.572,E2 6734.572} C_VEL
LIN {X 0,Y 474.102,Z 776.102,A -85,B 0,C 180,E1 6738.527,E2 6738.527} C_VEL
LIN {X 0,Y 473.701,Z 786.819,A -85,B 0,C 180,E1 6742.68,E2 6742.68} C_VEL
LIN {X 0,Y 473.629,Z 792.174,A -85,B 0,C 180,E1 6746.347,E2 6746.347} C_VEL
LIN {X 0,Y 473.527,Z 794,A -85,B 0,C 180,E1 6750.001,E2 6750.001} C_VEL
LIN {X 0,Y 473.634,Z 791.191,A -85,B 0,C 180,E1 6754.569,E2 6754.569} C_VEL
LIN {X 0,Y 473.863,Z 782.572,A -85,B 0,C 180,E1 6759.205,E2 6759.205} C_VEL
LIN {X 0,Y 474.436,Z 769.817,A -85,B 0,C 180,E1 6763.228,E2 6763.228} C_VEL
LIN {X 0,Y 475.681,Z 750.952,A -85,B 0,C 180,E1 6767.305,E2 6767.305} C_VEL
LIN {X 0,Y 477.675,Z 726.17,A -85,B 0,C 180,E1 6771.16,E2 6771.16} C_VEL
LIN {X 0,Y 480.24,Z 698.034,A -85,B 0,C 180,E1 6774.389,E2 6774.389} C_VEL
LIN {X 0,Y 483.044,Z 664.823,A -85,B 0,C 180,E1 6777.191,E2 6777.191} C_VEL
LIN {X 0,Y 485.578,Z 629.64,A -85,B 0,C 180,E1 6779.261,E2 6779.261} C_VEL
LIN {X 0,Y 487.566,Z 593.026,A -85,B 0,C 180,E1 6780.651,E2 6780.651} C_VEL
LIN {X 0,Y 487.609,Z 567.508,A -85,B 0,C 180,E1 6781.267,E2 6781.267} C_VEL
LIN {X 0,Y 472.664,Z 529.66,A -85,B 0,C 180,E1 6782.997,E2 6782.997} C_VEL
LIN {X 0,Y 472.653,Z 529.66,A -85,B 0,C 180,E1 6787.345,E2 6787.345} C_VEL
LIN {X 0,Y 472.477,Z 529.66,A -85,B 0,C 180,E1 6792.733,E2 6792.733} C_VEL
LIN {X 0,Y 472.486,Z 529.66,A -85,B 0,C 180,E1 6797.884,E2 6797.884} C_VEL
LIN {X 0,Y 472.645,Z 529.66,A -85,B 0,C 180,E1 6802.956,E2 6802.956} C_VEL
LIN {X 0,Y 472.628,Z 529.66,A -85,B 0,C 180,E1 6809.549,E2 6809.549} C_VEL
LIN {X 0,Y 472.766,Z 529.66,A -85,B 0,C 180,E1 6815.488,E2 6815.488} C_VEL
LIN {X 0,Y 472.959,Z 529.66,A -85,B 0,C 180,E1 6821.397,E2 6821.397} C_VEL
LIN {X 0,Y 472.903,Z 529.66,A -85,B 0,C 180,E1 6827.096,E2 6827.096} C_VEL
LIN {X 0,Y 473.198,Z 529.66,A -85,B 0,C 180,E1 6832.674,E2 6832.674} C_VEL
LIN {X 0,Y 473.512,Z 529.66,A -85,B 0,C 180,E1 6838.176,E2 6838.176} C_VEL
LIN {X 0,Y 473.389,Z 529.66,A -85,B 0,C 180,E1 6843.658,E2 6843.658} C_VEL
LIN {X 0,Y 473.157,Z 529.66,A -85,B 0,C 180,E1 6849.178,E2 6849.178} C_VEL
LIN {X 0,Y 473.041,Z 529.66,A -85,B 0,C 180,E1 6854.788,E2 6854.788} C_VEL
LIN {X 0,Y 472.875,Z 529.66,A -85,B 0,C 180,E1 6860.552,E2 6860.552} C_VEL
LIN {X 0,Y 472.649,Z 529.66,A -85,B 0,C 180,E1 6866.626,E2 6866.626} C_VEL
LIN {X 0,Y 472.533,Z 529.66,A -85,B 0,C 180,E1 6872.882,E2 6872.882} C_VEL
LIN {X 0,Y 472.487,Z 529.66,A -85,B 0,C 180,E1 6877.361,E2 6877.361} C_VEL
LIN {X 0,Y 472.746,Z 529.66,A -85,B 0,C 180,E1 6884.609,E2 6884.609} C_VEL
LIN {X 0,Y 479.962,Z 555.022,A -85,B 0,C 180,E1 6885.365,E2 6885.365} C_VEL
LIN {X 0,Y 479.345,Z 628.075,A -85,B 0,C 180,E1 6886.605,E2 6886.605} C_VEL
LIN {X 0,Y 478.339,Z 656.89,A -85,B 0,C 180,E1 6887.829,E2 6887.829} C_VEL
LIN {X 0,Y 477.027,Z 682.847,A -85,B 0,C 180,E1 6889.689,E2 6889.689} C_VEL
LIN {X 0,Y 475.674,Z 705.168,A -85,B 0,C 180,E1 6892.113,E2 6892.113} C_VEL
LIN {X 0,Y 474.643,Z 723.56,A -85,B 0,C 180,E1 6895.091,E2 6895.091} C_VEL
LIN {X 0,Y 474.068,Z 736.426,A -85,B 0,C 180,E1 6898.313,E2 6898.313} C_VEL
LIN {X 0,Y 473.743,Z 743.61,A -85,B 0,C 180,E1 6901.458,E2 6901.458} C_VEL
LIN {X 0,Y 473.46,Z 745.824,A -85,B 0,C 180,E1 6903.499,E2 6903.499} C_VEL
LIN {X 0,Y 473.377,Z 746.204,A -85,B 0,C 180,E1 6905.517,E2 6905.517} C_VEL
LIN {X 0,Y 473.679,Z 743.451,A -85,B 0,C 180,E1 6908.523,E2 6908.523} C_VEL
LIN {X 0,Y 474.108,Z 734.641,A -85,B 0,C 180,E1 6912.124,E2 6912.124} C_VEL
LIN {X 0,Y 474.809,Z 721.133,A -85,B 0,C 180,E1 6915.27,E2 6915.27} C_VEL
LIN {X 0,Y 475.83,Z 702.603,A -85,B 0,C 180,E1 6918.103,E2 6918.103} C_VEL
LIN {X 0,Y 477.18,Z 679.804,A -85,B 0,C 180,E1 6920.465,E2 6920.465} C_VEL
LIN {X 0,Y 478.464,Z 653.84,A -85,B 0,C 180,E1 6922.239,E2 6922.239} C_VEL
LIN {X 0,Y 479.4,Z 625.015,A -85,B 0,C 180,E1 6923.38,E2 6923.38} C_VEL
LIN {X 0,Y 479.281,Z 552.445,A -85,B 0,C 180,E1 6924.608,E2 6924.608} C_VEL
LIN {X 0,Y 473.118,Z 529.66,A -85,B 0,C 180,E1 6925.311,E2 6925.311} C_VEL
LIN {X 0,Y 473.523,Z 529.66,A -85,B 0,C 180,E1 6931.825,E2 6931.825} C_VEL
LIN {X 0,Y 473.225,Z 529.66,A -85,B 0,C 180,E1 6937.327,E2 6937.327} C_VEL
LIN {X 0,Y 473.019,Z 529.66,A -85,B 0,C 180,E1 6942.903,E2 6942.903} C_VEL
LIN {X 0,Y 472.894,Z 529.66,A -85,B 0,C 180,E1 6948.607,E2 6948.607} C_VEL
LIN {X 0,Y 472.744,Z 529.66,A -85,B 0,C 180,E1 6954.516,E2 6954.516} C_VEL
LIN {X 0,Y 472.538,Z 529.66,A -85,B 0,C 180,E1 6960.726,E2 6960.726} C_VEL
LIN {X 0,Y 472.666,Z 529.66,A -85,B 0,C 180,E1 6967.341,E2 6967.341} C_VEL
LIN {X 0,Y 472.479,Z 529.66,A -85,B 0,C 180,E1 6972.726,E2 6972.726} C_VEL
LIN {X 0,Y 472.472,Z 529.66,A -85,B 0,C 180,E1 6977.876,E2 6977.876} C_VEL
LIN {X 0,Y 472.577,Z 529.66,A -85,B 0,C 180,E1 6982.965,E2 6982.965} C_VEL
LIN {X 0,Y 472.58,Z 529.66,A -85,B 0,C 180,E1 6989.556,E2 6989.556} C_VEL
LIN {X 0,Y 472.713,Z 529.66,A -85,B 0,C 180,E1 6992.124,E2 6992.124} C_VEL
LIN {X 0,Y 484.943,Z 564.4,A -85,B 0,C 180,E1 6993.506,E2 6993.506} C_VEL
LIN {X 0,Y 483.501,Z 598.113,A -85,B 0,C 180,E1 6994.622,E2 6994.622} C_VEL
LIN {X 0,Y 481.405,Z 631,A -85,B 0,C 180,E1 6996.441,E2 6996.441} C_VEL
LIN {X 0,Y 479.027,Z 661.135,A -85,B 0,C 180,E1 6998.899,E2 6998.899} C_VEL
LIN {X 0,Y 476.911,Z 686.45,A -85,B 0,C 180,E1 7001.805,E2 7001.805} C_VEL
LIN {X 0,Y 475.255,Z 708.322,A -85,B 0,C 180,E1 7005.283,E2 7005.283} C_VEL
LIN {X 0,Y 474.199,Z 724.695,A -85,B 0,C 180,E1 7008.991,E2 7008.991} C_VEL
LIN {X 0,Y 473.786,Z 735.618,A -85,B 0,C 180,E1 7012.678,E2 7012.678} C_VEL
LIN {X 0,Y 473.659,Z 741.918,A -85,B 0,C 180,E1 7016.344,E2 7016.344} C_VEL
LIN {X 0,Y 473.548,Z 743.998,A -85,B 0,C 180,E1 7019.998,E2 7019.998} C_VEL
LIN {X 0,Y 473.667,Z 741.825,A -85,B 0,C 180,E1 7023.651,E2 7023.651} C_VEL
LIN {X 0,Y 473.879,Z 734.315,A -85,B 0,C 180,E1 7027.775,E2 7027.775} C_VEL
LIN {X 0,Y 474.471,Z 720.902,A -85,B 0,C 180,E1 7031.928,E2 7031.928} C_VEL
LIN {X 0,Y 475.723,Z 702.792,A -85,B 0,C 180,E1 7035.639,E2 7035.639} C_VEL
LIN {X 0,Y 477.477,Z 680.301,A -85,B 0,C 180,E1 7038.898,E2 7038.898} C_VEL
LIN {X 0,Y 479.586,Z 653.484,A -85,B 0,C 180,E1 7041.707,E2 7041.707} C_VEL
LIN {X 0,Y 481.766,Z 623.694,A -85,B 0,C 180,E1 7043.903,E2 7043.903} C_VEL
LIN {X 0,Y 483.626,Z 590.32,A -85,B 0,C 180,E1 7045.553,E2 7045.553} C_VEL
LIN {X 0,Y 484.142,Z 561.564,A -85,B 0,C 180,E1 7046.434,E2 7046.434} C_VEL
LIN {X 0,Y 472.728,Z 529.66,A -85,B 0,C 180,E1 7047.721,E2 7047.721} C_VEL
LIN {X 0,Y 472.547,Z 529.66,A -85,B 0,C 180,E1 7053.876,E2 7053.876} C_VEL
LIN {X 0,Y 472.412,Z 529.66,A -85,B 0,C 180,E1 7059.95,E2 7059.95} C_VEL
LIN {X 0,Y 472.44,Z 529.66,A -85,B 0,C 180,E1 7065.116,E2 7065.116} C_VEL
LIN {X 0,Y 469.937,Z 529.66,A -85,B 0,C 180,E1 7066.681,E2 7066.681} C_VEL
LIN {X 0,Y 464.644,Z 529.66,A -85,B 0,C 180,E1 7069.031,E2 7069.031} C_VEL
LIN {X 0,Y 464.568,Z 529.66,A -85,B 0,C 180,E1 7069.302,E2 7069.302} C_VEL
LIN {X 0,Y 464.676,Z 529.66,A -85,B 0,C 180,E1 7074.272,E2 7074.272} C_VEL
LIN {X 0,Y 464.734,Z 529.66,A -85,B 0,C 180,E1 7077.186,E2 7077.186} C_VEL
LIN {X 0,Y 479.631,Z 570.842,A -85,B 0,C 180,E1 7078.801,E2 7078.801} C_VEL
LIN {X 0,Y 478.361,Z 608.63,A -85,B 0,C 180,E1 7079.811,E2 7079.811} C_VEL
LIN {X 0,Y 476.312,Z 645.721,A -85,B 0,C 180,E1 7081.535,E2 7081.535} C_VEL
LIN {X 0,Y 473.719,Z 680.026,A -85,B 0,C 180,E1 7083.898,E2 7083.898} C_VEL
LIN {X 0,Y 471.172,Z 711.243,A -85,B 0,C 180,E1 7086.905,E2 7086.905} C_VEL
LIN {X 0,Y 468.917,Z 738.386,A -85,B 0,C 180,E1 7090.497,E2 7090.497} C_VEL
LIN {X 0,Y 467.123,Z 760.632,A -85,B 0,C 180,E1 7094.544,E2 7094.544} C_VEL
LIN {X 0,Y 466.168,Z 777.036,A -85,B 0,C 180,E1 7098.802,E2 7098.802} C_VEL
LIN {X 0,Y 465.81,Z 786.613,A -85,B 0,C 180,E1 7102.555,E2 7102.555} C_VEL
LIN {X 0,Y 465.739,Z 792.148,A -85,B 0,C 180,E1 7106.285,E2 7106.285} C_VEL
LIN {X 0,Y 465.637,Z 793.998,A -85,B 0,C 180,E1 7110.001,E2 7110.001} C_VEL
LIN {X 0,Y 465.761,Z 792.149,A -85,B 0,C 180,E1 7113.716,E2 7113.716} C_VEL
LIN {X 0,Y 465.955,Z 784.859,A -85,B 0,C 180,E1 7118.284,E2 7118.284} C_VEL
LIN {X 0,Y 466.404,Z 772.43,A -85,B 0,C 180,E1 7122.615,E2 7122.615} C_VEL
LIN {X 0,Y 467.627,Z 754.039,A -85,B 0,C 180,E1 7126.884,E2 7126.884} C_VEL
LIN {X 0,Y 469.548,Z 731.234,A -85,B 0,C 180,E1 7130.703,E2 7130.703} C_VEL
LIN {X 0,Y 472.184,Z 703.267,A -85,B 0,C 180,E1 7134.172,E2 7134.172} C_VEL
LIN {X 0,Y 475.136,Z 670.783,A -85,B 0,C 180,E1 7137.104,E2 7137.104} C_VEL
LIN {X 0,Y 477.93,Z 636.095,A -85,B 0,C 180,E1 7139.331,E2 7139.331} C_VEL
LIN {X 0,Y 480.164,Z 598.528,A -85,B 0,C 180,E1 7140.909,E2 7140.909} C_VEL
LIN {X 0,Y 480.729,Z 570.101,A -85,B 0,C 180,E1 7141.637,E2 7141.637} C_VEL
LIN {X 0,Y 464.724,Z 529.66,A -85,B 0,C 180,E1 7143.505,E2 7143.505} C_VEL
LIN {X 0,Y 464.566,Z 529.66,A -85,B 0,C 180,E1 7150.515,E2 7150.515} C_VEL
LIN {X 0,Y 464.586,Z 529.66,A -85,B 0,C 180,E1 7156.997,E2 7156.997} C_VEL
LIN {X 0,Y 464.628,Z 529.66,A -85,B 0,C 180,E1 7161.901,E2 7161.901} C_VEL
LIN {X 0,Y 464.591,Z 529.66,A -85,B 0,C 180,E1 7167.618,E2 7167.618} C_VEL
LIN {X 0,Y 464.766,Z 529.66,A -85,B 0,C 180,E1 7172.967,E2 7172.967} C_VEL
LIN {X 0,Y 464.966,Z 529.66,A -85,B 0,C 180,E1 7179.087,E2 7179.087} C_VEL
LIN {X 0,Y 464.91,Z 529.66,A -85,B 0,C 180,E1 7184.953,E2 7184.953} C_VEL
LIN {X 0,Y 465.142,Z 529.66,A -85,B 0,C 180,E1 7190.668,E2 7190.668} C_VEL
LIN {X 0,Y 465.395,Z 529.66,A -85,B 0,C 180,E1 7196.284,E2 7196.284} C_VEL
LIN {X 0,Y 465.438,Z 529.66,A -85,B 0,C 180,E1 7201.86,E2 7201.86} C_VEL
LIN {X 0,Y 465.263,Z 529.66,A -85,B 0,C 180,E1 7207.457,E2 7207.457} C_VEL
LIN {X 0,Y 465.165,Z 529.66,A -85,B 0,C 180,E1 7213.292,E2 7213.292} C_VEL
LIN {X 0,Y 464.948,Z 529.66,A -85,B 0,C 180,E1 7219.744,E2 7219.744} C_VEL
LIN {X 0,Y 464.784,Z 529.66,A -85,B 0,C 180,E1 7224.967,E2 7224.967} C_VEL
LIN {X 0,Y 464.625,Z 529.66,A -85,B 0,C 180,E1 7231.311,E2 7231.311} C_VEL
LIN {X 0,Y 464.596,Z 529.66,A -85,B 0,C 180,E1 7235.78,E2 7235.78} C_VEL
LIN {X 0,Y 464.614,Z 529.66,A -85,B 0,C 180,E1 7243.006,E2 7243.006} C_VEL
LIN {X 0,Y 464.771,Z 529.66,A -85,B 0,C 180,E1 7244.262,E2 7244.262} C_VEL
LIN {X 0,Y 472.581,Z 557.027,A -85,B 0,C 180,E1 7245.074,E2 7245.074} C_VEL
LIN {X 0,Y 471.858,Z 628.359,A -85,B 0,C 180,E1 7246.303,E2 7246.303} C_VEL
LIN {X 0,Y 470.817,Z 656.327,A -85,B 0,C 180,E1 7247.493,E2 7247.493} C_VEL
LIN {X 0,Y 469.501,Z 681.98,A -85,B 0,C 180,E1 7249.328,E2 7249.328} C_VEL
LIN {X 0,Y 468.007,Z 704.709,A -85,B 0,C 180,E1 7251.784,E2 7251.784} C_VEL
LIN {X 0,Y 466.865,Z 723.46,A -85,B 0,C 180,E1 7254.827,E2 7254.827} C_VEL
LIN {X 0,Y 466.261,Z 736.316,A -85,B 0,C 180,E1 7258.045,E2 7258.045} C_VEL
LIN {X 0,Y 465.909,Z 743.328,A -85,B 0,C 180,E1 7260.987,E2 7260.987} C_VEL
LIN {X 0,Y 465.638,Z 745.88,A -85,B 0,C 180,E1 7263.018,E2 7263.018} C_VEL
LIN {X 0,Y 465.488,Z 746.651,A -85,B 0,C 180,E1 7265.192,E2 7265.192} C_VEL
LIN {X 0,Y 465.735,Z 744.43,A -85,B 0,C 180,E1 7268.183,E2 7268.183} C_VEL
LIN {X 0,Y 466.174,Z 736.601,A -85,B 0,C 180,E1 7271.748,E2 7271.748} C_VEL
LIN {X 0,Y 466.949,Z 722.54,A -85,B 0,C 180,E1 7275.236,E2 7275.236} C_VEL
LIN {X 0,Y 468.051,Z 704.401,A -85,B 0,C 180,E1 7278.139,E2 7278.139} C_VEL
LIN {X 0,Y 469.531,Z 680.921,A -85,B 0,C 180,E1 7280.652,E2 7280.652} C_VEL
LIN {X 0,Y 470.932,Z 654.201,A -85,B 0,C 180,E1 7282.52,E2 7282.52} C_VEL
LIN {X 0,Y 471.93,Z 625.119,A -85,B 0,C 180,E1 7283.684,E2 7283.684} C_VEL
LIN {X 0,Y 471.885,Z 553.93,A -85,B 0,C 180,E1 7284.906,E2 7284.906} C_VEL
LIN {X 0,Y 465.28,Z 529.66,A -85,B 0,C 180,E1 7285.699,E2 7285.699} C_VEL
LIN {X 0,Y 465.62,Z 529.66,A -85,B 0,C 180,E1 7291.856,E2 7291.856} C_VEL
LIN {X 0,Y 465.319,Z 529.66,A -85,B 0,C 180,E1 7297.452,E2 7297.452} C_VEL
LIN {X 0,Y 465.066,Z 529.66,A -85,B 0,C 180,E1 7303.236,E2 7303.236} C_VEL
LIN {X 0,Y 464.915,Z 529.66,A -85,B 0,C 180,E1 7309.73,E2 7309.73} C_VEL
LIN {X 0,Y 464.767,Z 529.66,A -85,B 0,C 180,E1 7314.965,E2 7314.965} C_VEL
LIN {X 0,Y 464.569,Z 529.66,A -85,B 0,C 180,E1 7321.311,E2 7321.311} C_VEL
LIN {X 0,Y 464.701,Z 529.66,A -85,B 0,C 180,E1 7325.767,E2 7325.767} C_VEL
LIN {X 0,Y 464.553,Z 529.66,A -85,B 0,C 180,E1 7331.657,E2 7331.657} C_VEL
LIN {X 0,Y 464.552,Z 529.66,A -85,B 0,C 180,E1 7338.339,E2 7338.339} C_VEL
LIN {X 0,Y 464.606,Z 529.66,A -85,B 0,C 180,E1 7344.288,E2 7344.288} C_VEL
LIN {X 0,Y 464.744,Z 529.66,A -85,B 0,C 180,E1 7351.242,E2 7351.242} C_VEL
LIN {X 0,Y 464.774,Z 529.66,A -85,B 0,C 180,E1 7351.618,E2 7351.618} C_VEL
LIN {X 0,Y 477.776,Z 565.415,A -85,B 0,C 180,E1 7353.127,E2 7353.127} C_VEL
LIN {X 0,Y 476.214,Z 599.803,A -85,B 0,C 180,E1 7354.307,E2 7354.307} C_VEL
LIN {X 0,Y 473.963,Z 632.436,A -85,B 0,C 180,E1 7356.173,E2 7356.173} C_VEL
LIN {X 0,Y 471.449,Z 662.089,A -85,B 0,C 180,E1 7358.655,E2 7358.655} C_VEL
LIN {X 0,Y 469.181,Z 687.998,A -85,B 0,C 180,E1 7361.705,E2 7361.705} C_VEL
LIN {X 0,Y 467.456,Z 709.531,A -85,B 0,C 180,E1 7365.233,E2 7365.233} C_VEL
LIN {X 0,Y 466.284,Z 726.618,A -85,B 0,C 180,E1 7369.273,E2 7369.273} C_VEL
LIN {X 0,Y 465.88,Z 737.785,A -85,B 0,C 180,E1 7373.488,E2 7373.488} C_VEL
LIN {X 0,Y 465.769,Z 742.014,A -85,B 0,C 180,E1 7376.282,E2 7376.282} C_VEL
LIN {X 0,Y 465.657,Z 744.06,A -85,B 0,C 180,E1 7379.998,E2 7379.998} C_VEL
LIN {X 0,Y 465.777,Z 741.937,A -85,B 0,C 180,E1 7383.713,E2 7383.713} C_VEL
LIN {X 0,Y 466.023,Z 734.65,A -85,B 0,C 180,E1 7387.879,E2 7387.879} C_VEL
LIN {X 0,Y 466.683,Z 721.2,A -85,B 0,C 180,E1 7392.13,E2 7392.13} C_VEL
LIN {X 0,Y 467.997,Z 702.985,A -85,B 0,C 180,E1 7395.904,E2 7395.904} C_VEL
LIN {X 0,Y 469.904,Z 680.317,A -85,B 0,C 180,E1 7399.215,E2 7399.215} C_VEL
LIN {X 0,Y 472.122,Z 653.489,A -85,B 0,C 180,E1 7402.046,E2 7402.046} C_VEL
LIN {X 0,Y 474.437,Z 623.088,A -85,B 0,C 180,E1 7404.295,E2 7404.295} C_VEL
LIN {X 0,Y 476.431,Z 589.355,A -85,B 0,C 180,E1 7405.959,E2 7405.959} C_VEL
LIN {X 0,Y 476.894,Z 563.469,A -85,B 0,C 180,E1 7406.775,E2 7406.775} C_VEL
LIN {X 0,Y 464.791,Z 529.66,A -85,B 0,C 180,E1 7408.254,E2 7408.254} C_VEL
LIN {X 0,Y 464.634,Z 529.66,A -85,B 0,C 180,E1 7413.508,E2 7413.508} C_VEL
LIN {X 0,Y 464.486,Z 529.66,A -85,B 0,C 180,E1 7418.769,E2 7418.769} C_VEL
LIN {X 0,Y 464.532,Z 529.66,A -85,B 0,C 180,E1 7425.61,E2 7425.61} C_VEL
LIN {X 0,Y 464.568,Z 529.66,A -85,B 0,C 180,E1 7429.302,E2 7429.302} C_VEL
LIN {X 0,Y 462.155,Z 529.66,A -85,B 0,C 180,E1 7430.894,E2 7430.894} C_VEL
LIN {X 0,Y 456.672,Z 529.66,A -85,B 0,C 180,E1 7433.56,E2 7433.56} C_VEL
LIN {X 0,Y 456.805,Z 529.66,A -85,B 0,C 180,E1 7436.638,E2 7436.638} C_VEL
LIN {X 0,Y 472.43,Z 574.531,A -85,B 0,C 180,E1 7438.479,E2 7438.479} C_VEL
LIN {X 0,Y 470.902,Z 612.211,A -85,B 0,C 180,E1 7439.577,E2 7439.577} C_VEL
LIN {X 0,Y 468.65,Z 648.681,A -85,B 0,C 180,E1 7441.376,E2 7441.376} C_VEL
LIN {X 0,Y 465.934,Z 682.599,A -85,B 0,C 180,E1 7443.816,E2 7443.816} C_VEL
LIN {X 0,Y 463.369,Z 712.374,A -85,B 0,C 180,E1 7446.797,E2 7446.797} C_VEL
LIN {X 0,Y 461.08,Z 738.905,A -85,B 0,C 180,E1 7450.401,E2 7450.401} C_VEL
LIN {X 0,Y 459.259,Z 760.977,A -85,B 0,C 180,E1 7454.517,E2 7454.517} C_VEL
LIN {X 0,Y 458.32,Z 776.429,A -85,B 0,C 180,E1 7458.607,E2 7458.607} C_VEL
LIN {X 0,Y 457.929,Z 786.098,A -85,B 0,C 180,E1 7462.427,E2 7462.427} C_VEL
LIN {X 0,Y 457.844,Z 791.704,A -85,B 0,C 180,E1 7466.221,E2 7466.221} C_VEL
LIN {X 0,Y 457.747,Z 793.6,A -85,B 0,C 180,E1 7470.001,E2 7470.001} C_VEL
LIN {X 0,Y 457.863,Z 791.729,A -85,B 0,C 180,E1 7473.78,E2 7473.78} C_VEL
LIN {X 0,Y 458.047,Z 784.928,A -85,B 0,C 180,E1 7478.175,E2 7478.175} C_VEL
LIN {X 0,Y 458.565,Z 771.905,A -85,B 0,C 180,E1 7482.834,E2 7482.834} C_VEL
LIN {X 0,Y 459.753,Z 754.65,A -85,B 0,C 180,E1 7486.936,E2 7486.936} C_VEL
LIN {X 0,Y 461.772,Z 732.135,A -85,B 0,C 180,E1 7490.817,E2 7490.817} C_VEL
LIN {X 0,Y 464.504,Z 704.448,A -85,B 0,C 180,E1 7494.352,E2 7494.352} C_VEL
LIN {X 0,Y 467.681,Z 671.775,A -85,B 0,C 180,E1 7497.392,E2 7497.392} C_VEL
LIN {X 0,Y 470.594,Z 637.602,A -85,B 0,C 180,E1 7499.65,E2 7499.65} C_VEL
LIN {X 0,Y 473.04,Z 599.85,A -85,B 0,C 180,E1 7501.297,E2 7501.297} C_VEL
LIN {X 0,Y 473.669,Z 572.351,A -85,B 0,C 180,E1 7502.035,E2 7502.035} C_VEL
LIN {X 0,Y 456.752,Z 529.66,A -85,B 0,C 180,E1 7504.035,E2 7504.035} C_VEL
LIN {X 0,Y 456.676,Z 529.66,A -85,B 0,C 180,E1 7510.542,E2 7510.542} C_VEL
LIN {X 0,Y 456.678,Z 529.66,A -85,B 0,C 180,E1 7516.632,E2 7516.632} C_VEL
LIN {X 0,Y 456.688,Z 529.66,A -85,B 0,C 180,E1 7522.469,E2 7522.469} C_VEL
LIN {X 0,Y 456.683,Z 529.66,A -85,B 0,C 180,E1 7529.217,E2 7529.217} C_VEL
LIN {X 0,Y 456.847,Z 529.66,A -85,B 0,C 180,E1 7534.574,E2 7534.574} C_VEL
LIN {X 0,Y 457.081,Z 529.66,A -85,B 0,C 180,E1 7540.726,E2 7540.726} C_VEL
LIN {X 0,Y 457.083,Z 529.66,A -85,B 0,C 180,E1 7546.641,E2 7546.641} C_VEL
LIN {X 0,Y 457.366,Z 529.66,A -85,B 0,C 180,E1 7552.419,E2 7552.419} C_VEL
LIN {X 0,Y 457.699,Z 529.66,A -85,B 0,C 180,E1 7558.113,E2 7558.113} C_VEL
LIN {X 0,Y 457.574,Z 529.66,A -85,B 0,C 180,E1 7563.784,E2 7563.784} C_VEL
LIN {X 0,Y 457.311,Z 529.66,A -85,B 0,C 180,E1 7569.499,E2 7569.499} C_VEL
LIN {X 0,Y 457.162,Z 529.66,A -85,B 0,C 180,E1 7575.314,E2 7575.314} C_VEL
LIN {X 0,Y 456.994,Z 529.66,A -85,B 0,C 180,E1 7581.3,E2 7581.3} C_VEL
LIN {X 0,Y 456.784,Z 529.66,A -85,B 0,C 180,E1 7587.55,E2 7587.55} C_VEL
LIN {X 0,Y 456.633,Z 529.66,A -85,B 0,C 180,E1 7594.293,E2 7594.293} C_VEL
LIN {X 0,Y 456.563,Z 529.66,A -85,B 0,C 180,E1 7600.519,E2 7600.519} C_VEL
LIN {X 0,Y 456.795,Z 529.66,A -85,B 0,C 180,E1 7603.885,E2 7603.885} C_VEL
LIN {X 0,Y 465.193,Z 559.616,A -85,B 0,C 180,E1 7604.782,E2 7604.782} C_VEL
LIN {X 0,Y 464.402,Z 628.772,A -85,B 0,C 180,E1 7605.995,E2 7605.995} C_VEL
LIN {X 0,Y 463.271,Z 657.24,A -85,B 0,C 180,E1 7607.232,E2 7607.232} C_VEL
LIN {X 0,Y 461.815,Z 683.797,A -85,B 0,C 180,E1 7609.193,E2 7609.193} C_VEL
LIN {X 0,Y 460.218,Z 706.588,A -85,B 0,C 180,E1 7611.769,E2 7611.769} C_VEL
LIN {X 0,Y 459.136,Z 723.428,A -85,B 0,C 180,E1 7614.569,E2 7614.569} C_VEL
LIN {X 0,Y 458.439,Z 736.458,A -85,B 0,C 180,E1 7617.848,E2 7617.848} C_VEL
LIN {X 0,Y 457.946,Z 744.682,A -85,B 0,C 180,E1 7621.529,E2 7621.529} C_VEL
LIN {X 0,Y 457.58,Z 747.024,A -85,B 0,C 180,E1 7624.613,E2 7624.613} C_VEL
LIN {X 0,Y 457.724,Z 745.824,A -85,B 0,C 180,E1 7627.386,E2 7627.386} C_VEL
LIN {X 0,Y 458.176,Z 739.967,A -85,B 0,C 180,E1 7630.77,E2 7630.77} C_VEL
LIN {X 0,Y 458.824,Z 728.288,A -85,B 0,C 180,E1 7634.256,E2 7634.256} C_VEL
LIN {X 0,Y 459.886,Z 711.172,A -85,B 0,C 180,E1 7637.444,E2 7637.444} C_VEL
LIN {X 0,Y 461.355,Z 689.926,A -85,B 0,C 180,E1 7640.096,E2 7640.096} C_VEL
LIN {X 0,Y 462.827,Z 665.299,A -85,B 0,C 180,E1 7642.152,E2 7642.152} C_VEL
LIN {X 0,Y 464.078,Z 637.629,A -85,B 0,C 180,E1 7643.592,E2 7643.592} C_VEL
LIN {X 0,Y 464.689,Z 608.313,A -85,B 0,C 180,E1 7644.348,E2 7644.348} C_VEL
LIN {X 0,Y 464.527,Z 555.583,A -85,B 0,C 180,E1 7645.208,E2 7645.208} C_VEL
LIN {X 0,Y 457.458,Z 529.66,A -85,B 0,C 180,E1 7646.067,E2 7646.067} C_VEL
LIN {X 0,Y 457.71,Z 529.66,A -85,B 0,C 180,E1 7651.888,E2 7651.888} C_VEL
LIN {X 0,Y 457.318,Z 529.66,A -85,B 0,C 180,E1 7658.139,E2 7658.139} C_VEL
LIN {X 0,Y 457.168,Z 529.66,A -85,B 0,C 180,E1 7663.358,E2 7663.358} C_VEL
LIN {X 0,Y 457.023,Z 529.66,A -85,B 0,C 180,E1 7669.279,E2 7669.279} C_VEL
LIN {X 0,Y 456.8,Z 529.66,A -85,B 0,C 180,E1 7675.431,E2 7675.431} C_VEL
LIN {X 0,Y 456.651,Z 529.66,A -85,B 0,C 180,E1 7681.918,E2 7681.918} C_VEL
LIN {X 0,Y 456.719,Z 529.66,A -85,B 0,C 180,E1 7688.884,E2 7688.884} C_VEL
LIN {X 0,Y 456.66,Z 529.66,A -85,B 0,C 180,E1 7693.941,E2 7693.941} C_VEL
LIN {X 0,Y 456.657,Z 529.66,A -85,B 0,C 180,E1 7699.465,E2 7699.465} C_VEL
LIN {X 0,Y 456.621,Z 529.66,A -85,B 0,C 180,E1 7705.817,E2 7705.817} C_VEL
LIN {X 0,Y 456.845,Z 529.66,A -85,B 0,C 180,E1 7711.082,E2 7711.082} C_VEL
LIN {X 0,Y 470.578,Z 567.026,A -85,B 0,C 180,E1 7712.751,E2 7712.751} C_VEL
LIN {X 0,Y 468.878,Z 601.6,A -85,B 0,C 180,E1 7713.992,E2 7713.992} C_VEL
LIN {X 0,Y 466.544,Z 633.872,A -85,B 0,C 180,E1 7715.897,E2 7715.897} C_VEL
LIN {X 0,Y 463.902,Z 663.021,A -85,B 0,C 180,E1 7718.401,E2 7718.401} C_VEL
LIN {X 0,Y 461.419,Z 689.995,A -85,B 0,C 180,E1 7721.666,E2 7721.666} C_VEL
LIN {X 0,Y 459.662,Z 710.7,A -85,B 0,C 180,E1 7725.182,E2 7725.182} C_VEL
LIN {X 0,Y 458.478,Z 726.887,A -85,B 0,C 180,E1 7729.089,E2 7729.089} C_VEL
LIN {X 0,Y 458.002,Z 738.155,A -85,B 0,C 180,E1 7733.376,E2 7733.376} C_VEL
LIN {X 0,Y 457.881,Z 742.419,A -85,B 0,C 180,E1 7736.218,E2 7736.218} C_VEL
LIN {X 0,Y 457.769,Z 744.483,A -85,B 0,C 180,E1 7739.997,E2 7739.997} C_VEL
LIN {X 0,Y 457.892,Z 742.38,A -85,B 0,C 180,E1 7743.777,E2 7743.777} C_VEL
LIN {X 0,Y 458.18,Z 734.503,A -85,B 0,C 180,E1 7748.244,E2 7748.244} C_VEL
LIN {X 0,Y 458.894,Z 721.497,A -85,B 0,C 180,E1 7752.339,E2 7752.339} C_VEL
LIN {X 0,Y 460.294,Z 703.169,A -85,B 0,C 180,E1 7756.177,E2 7756.177} C_VEL
LIN {X 0,Y 462.329,Z 680.304,A -85,B 0,C 180,E1 7759.542,E2 7759.542} C_VEL
LIN {X 0,Y 464.69,Z 653.325,A -85,B 0,C 180,E1 7762.409,E2 7762.409} C_VEL
LIN {X 0,Y 467.154,Z 622.502,A -85,B 0,C 180,E1 7764.699,E2 7764.699} C_VEL
LIN {X 0,Y 469.258,Z 587.938,A -85,B 0,C 180,E1 7766.401,E2 7766.401} C_VEL
LIN {X 0,Y 469.55,Z 565.006,A -85,B 0,C 180,E1 7767.152,E2 7767.152} C_VEL
LIN {X 0,Y 456.849,Z 529.66,A -85,B 0,C 180,E1 7768.814,E2 7768.814} C_VEL
LIN {X 0,Y 456.654,Z 529.66,A -85,B 0,C 180,E1 7774.3,E2 7774.3} C_VEL
LIN {X 0,Y 456.571,Z 529.66,A -85,B 0,C 180,E1 7780.523,E2 7780.523} C_VEL
LIN {X 0,Y 456.668,Z 529.66,A -85,B 0,C 180,E1 7786.627,E2 7786.627} C_VEL
LIN {X 0,Y 456.689,Z 529.66,A -85,B 0,C 180,E1 7792.462,E2 7792.462} C_VEL
LIN {X 0,Y 456.672,Z 529.66,A -85,B 0,C 180,E1 7793.56,E2 7793.56} C_VEL
LIN {X 0,Y 452.659,Z 529.66,A -85,B 0,C 180,E1 7794.496,E2 7794.496} C_VEL
LIN {X 0,Y 448.767,Z 529.66,A -85,B 0,C 180,E1 7795.448,E2 7795.448} C_VEL
LIN {X 0,Y 448.829,Z 529.66,A -85,B 0,C 180,E1 7796.044,E2 7796.044} C_VEL
LIN {X 0,Y 465.084,Z 574.702,A -85,B 0,C 180,E1 7798.057,E2 7798.057} C_VEL
LIN {X 0,Y 463.52,Z 614.285,A -85,B 0,C 180,E1 7799.278,E2 7799.278} C_VEL
LIN {X 0,Y 461.147,Z 650.466,A -85,B 0,C 180,E1 7801.135,E2 7801.135} C_VEL
LIN {X 0,Y 458.15,Z 685.033,A -85,B 0,C 180,E1 7803.732,E2 7803.732} C_VEL
LIN {X 0,Y 455.48,Z 714.727,A -85,B 0,C 180,E1 7806.834,E2 7806.834} C_VEL
LIN {X 0,Y 453.048,Z 740.955,A -85,B 0,C 180,E1 7810.545,E2 7810.545} C_VEL
LIN {X 0,Y 451.386,Z 761.282,A -85,B 0,C 180,E1 7814.489,E2 7814.489} C_VEL
LIN {X 0,Y 450.398,Z 777.247,A -85,B 0,C 180,E1 7818.894,E2 7818.894} C_VEL
LIN {X 0,Y 450.049,Z 787.372,A -85,B 0,C 180,E1 7823.261,E2 7823.261} C_VEL
LIN {X 0,Y 449.95,Z 791.257,A -85,B 0,C 180,E1 7826.155,E2 7826.155} C_VEL
LIN {X 0,Y 449.873,Z 793.178,A -85,B 0,C 180,E1 7830.001,E2 7830.001} C_VEL
LIN {X 0,Y 449.966,Z 791.306,A -85,B 0,C 180,E1 7833.847,E2 7833.847} C_VEL
LIN {X 0,Y 450.142,Z 784.472,A -85,B 0,C 180,E1 7838.32,E2 7838.32} C_VEL
LIN {X 0,Y 450.727,Z 771.373,A -85,B 0,C 180,E1 7843.062,E2 7843.062} C_VEL
LIN {X 0,Y 452.006,Z 754.023,A -85,B 0,C 180,E1 7847.236,E2 7847.236} C_VEL
LIN {X 0,Y 454.11,Z 731.386,A -85,B 0,C 180,E1 7851.185,E2 7851.185} C_VEL
LIN {X 0,Y 457.012,Z 704.066,A -85,B 0,C 180,E1 7854.716,E2 7854.716} C_VEL
LIN {X 0,Y 460.29,Z 672.183,A -85,B 0,C 180,E1 7857.736,E2 7857.736} C_VEL
LIN {X 0,Y 463.446,Z 637.447,A -85,B 0,C 180,E1 7860.071,E2 7860.071} C_VEL
LIN {X 0,Y 465.97,Z 600.22,A -85,B 0,C 180,E1 7861.725,E2 7861.725} C_VEL
LIN {X 0,Y 466.588,Z 574.315,A -85,B 0,C 180,E1 7862.452,E2 7862.452} C_VEL
LIN {X 0,Y 448.795,Z 529.66,A -85,B 0,C 180,E1 7864.61,E2 7864.61} C_VEL
LIN {X 0,Y 448.75,Z 529.66,A -85,B 0,C 180,E1 7869.711,E2 7869.711} C_VEL
LIN {X 0,Y 448.678,Z 529.66,A -85,B 0,C 180,E1 7875.072,E2 7875.072} C_VEL
LIN {X 0,Y 448.77,Z 529.66,A -85,B 0,C 180,E1 7880.659,E2 7880.659} C_VEL
LIN {X 0,Y 448.708,Z 529.66,A -85,B 0,C 180,E1 7887.451,E2 7887.451} C_VEL
LIN {X 0,Y 448.928,Z 529.66,A -85,B 0,C 180,E1 7894.092,E2 7894.092} C_VEL
LIN {X 0,Y 449.125,Z 529.66,A -85,B 0,C 180,E1 7900.371,E2 7900.371} C_VEL
LIN {X 0,Y 449.171,Z 529.66,A -85,B 0,C 180,E1 7906.975,E2 7906.975} C_VEL
LIN {X 0,Y 449.452,Z 529.66,A -85,B 0,C 180,E1 7912.285,E2 7912.285} C_VEL
LIN {X 0,Y 449.815,Z 529.66,A -85,B 0,C 180,E1 7918.08,E2 7918.08} C_VEL
LIN {X 0,Y 449.659,Z 529.66,A -85,B 0,C 180,E1 7923.851,E2 7923.851} C_VEL
LIN {X 0,Y 449.383,Z 529.66,A -85,B 0,C 180,E1 7929.668,E2 7929.668} C_VEL
LIN {X 0,Y 449.262,Z 529.66,A -85,B 0,C 180,E1 7935.59,E2 7935.59} C_VEL
LIN {X 0,Y 449.06,Z 529.66,A -85,B 0,C 180,E1 7941.696,E2 7941.696} C_VEL
LIN {X 0,Y 448.8,Z 529.66,A -85,B 0,C 180,E1 7948.083,E2 7948.083} C_VEL
LIN {X 0,Y 448.666,Z 529.66,A -85,B 0,C 180,E1 7954.876,E2 7954.876} C_VEL
LIN {X 0,Y 448.645,Z 529.66,A -85,B 0,C 180,E1 7959.724,E2 7959.724} C_VEL
LIN {X 0,Y 448.872,Z 530.304,A -85,B 0,C 180,E1 7963.501,E2 7963.501} C_VEL
LIN {X 0,Y 457.787,Z 560.701,A -85,B 0,C 180,E1 7964.453,E2 7964.453} C_VEL
LIN {X 0,Y 456.942,Z 629.567,A -85,B 0,C 180,E1 7965.688,E2 7965.688} C_VEL
LIN {X 0,Y 455.745,Z 658.95,A -85,B 0,C 180,E1 7967.012,E2 7967.012} C_VEL
LIN {X 0,Y 454.138,Z 685.252,A -85,B 0,C 180,E1 7969.021,E2 7969.021} C_VEL
LIN {X 0,Y 452.418,Z 708.179,A -85,B 0,C 180,E1 7971.711,E2 7971.711} C_VEL
LIN {X 0,Y 451.29,Z 724.931,A -85,B 0,C 180,E1 7974.62,E2 7974.62} C_VEL
LIN {X 0,Y 450.529,Z 737.668,A -85,B 0,C 180,E1 7977.989,E2 7977.989} C_VEL
LIN {X 0,Y 450.179,Z 743.777,A -85,B 0,C 180,E1 7980.639,E2 7980.639} C_VEL
LIN {X 0,Y 449.729,Z 747.331,A -85,B 0,C 180,E1 7984.138,E2 7984.138} C_VEL
LIN {X 0,Y 449.694,Z 747.084,A -85,B 0,C 180,E1 7986.254,E2 7986.254} C_VEL
LIN {X 0,Y 450.167,Z 742.648,A -85,B 0,C 180,E1 7989.82,E2 7989.82} C_VEL
LIN {X 0,Y 450.749,Z 732.423,A -85,B 0,C 180,E1 7993.471,E2 7993.471} C_VEL
LIN {X 0,Y 451.742,Z 717.249,A -85,B 0,C 180,E1 7996.723,E2 7996.723} C_VEL
LIN {X 0,Y 453.275,Z 696.344,A -85,B 0,C 180,E1 7999.685,E2 7999.685} C_VEL
LIN {X 0,Y 454.955,Z 671.542,A -85,B 0,C 180,E1 8002.016,E2 8002.016} C_VEL
LIN {X 0,Y 456.385,Z 643.566,A -85,B 0,C 180,E1 8003.67,E2 8003.67} C_VEL
LIN {X 0,Y 457.227,Z 614.73,A -85,B 0,C 180,E1 8004.566,E2 8004.566} C_VEL
LIN {X 0,Y 457.016,Z 556.601,A -85,B 0,C 180,E1 8005.537,E2 8005.537} C_VEL
LIN {X 0,Y 449.584,Z 529.66,A -85,B 0,C 180,E1 8006.391,E2 8006.391} C_VEL
LIN {X 0,Y 449.826,Z 529.66,A -85,B 0,C 180,E1 8011.922,E2 8011.922} C_VEL
LIN {X 0,Y 449.474,Z 529.66,A -85,B 0,C 180,E1 8017.717,E2 8017.717} C_VEL
LIN {X 0,Y 449.243,Z 529.66,A -85,B 0,C 180,E1 8023.598,E2 8023.598} C_VEL
LIN {X 0,Y 449.06,Z 529.66,A -85,B 0,C 180,E1 8029.792,E2 8029.792} C_VEL
LIN {X 0,Y 448.883,Z 529.66,A -85,B 0,C 180,E1 8035.913,E2 8035.913} C_VEL
LIN {X 0,Y 448.691,Z 529.66,A -85,B 0,C 180,E1 8042.774,E2 8042.774} C_VEL
LIN {X 0,Y 448.776,Z 529.66,A -85,B 0,C 180,E1 8049.34,E2 8049.34} C_VEL
LIN {X 0,Y 448.684,Z 529.66,A -85,B 0,C 180,E1 8055.066,E2 8055.066} C_VEL
LIN {X 0,Y 448.741,Z 529.66,A -85,B 0,C 180,E1 8060.661,E2 8060.661} C_VEL
LIN {X 0,Y 448.662,Z 529.66,A -85,B 0,C 180,E1 8067.441,E2 8067.441} C_VEL
LIN {X 0,Y 448.859,Z 530.261,A -85,B 0,C 180,E1 8070.596,E2 8070.596} C_VEL
LIN {X 0,Y 463.368,Z 569.993,A -85,B 0,C 180,E1 8072.399,E2 8072.399} C_VEL
LIN {X 0,Y 461.429,Z 605.072,A -85,B 0,C 180,E1 8073.754,E2 8073.754} C_VEL
LIN {X 0,Y 458.965,Z 636.915,A -85,B 0,C 180,E1 8075.731,E2 8075.731} C_VEL
LIN {X 0,Y 456.159,Z 666.412,A -85,B 0,C 180,E1 8078.399,E2 8078.399} C_VEL
LIN {X 0,Y 453.601,Z 692.039,A -85,B 0,C 180,E1 8081.649,E2 8081.649} C_VEL
LIN {X 0,Y 451.701,Z 713.433,A -85,B 0,C 180,E1 8085.454,E2 8085.454} C_VEL
LIN {X 0,Y 450.554,Z 728.695,A -85,B 0,C 180,E1 8089.383,E2 8089.383} C_VEL
LIN {X 0,Y 450.137,Z 738.514,A -85,B 0,C 180,E1 8093.259,E2 8093.259} C_VEL
LIN {X 0,Y 449.995,Z 742.823,A -85,B 0,C 180,E1 8096.152,E2 8096.152} C_VEL
LIN {X 0,Y 449.895,Z 744.905,A -85,B 0,C 180,E1 8099.997,E2 8099.997} C_VEL
LIN {X 0,Y 450.008,Z 742.823,A -85,B 0,C 180,E1 8103.843,E2 8103.843} C_VEL
LIN {X 0,Y 450.325,Z 735.202,A -85,B 0,C 180,E1 8108.254,E2 8108.254} C_VEL
LIN {X 0,Y 451.108,Z 721.793,A -85,B 0,C 180,E1 8112.555,E2 8112.555} C_VEL
LIN {X 0,Y 452.594,Z 703.343,A -85,B 0,C 180,E1 8116.46,E2 8116.46} C_VEL
LIN {X 0,Y 454.771,Z 680.279,A -85,B 0,C 180,E1 8119.881,E2 8119.881} C_VEL
LIN {X 0,Y 457.394,Z 652.214,A -85,B 0,C 180,E1 8122.862,E2 8122.862} C_VEL
LIN {X 0,Y 460.048,Z 620.132,A -85,B 0,C 180,E1 8125.237,E2 8125.237} C_VEL
LIN {X 0,Y 462.225,Z 585.738,A -85,B 0,C 180,E1 8126.895,E2 8126.895} C_VEL
LIN {X 0,Y 462.412,Z 567.131,A -85,B 0,C 180,E1 8127.522,E2 8127.522} C_VEL
LIN {X 0,Y 448.901,Z 529.66,A -85,B 0,C 180,E1 8129.408,E2 8129.408} C_VEL
LIN {X 0,Y 448.673,Z 529.66,A -85,B 0,C 180,E1 8136.181,E2 8136.181} C_VEL
LIN {X 0,Y 448.634,Z 529.66,A -85,B 0,C 180,E1 8142.272,E2 8142.272} C_VEL
LIN {X 0,Y 448.706,Z 529.66,A -85,B 0,C 180,E1 8147.733,E2 8147.733} C_VEL
LIN {X 0,Y 448.742,Z 529.66,A -85,B 0,C 180,E1 8153.803,E2 8153.803} C_VEL
LIN {X 0,Y 448.767,Z 529.66,A -85,B 0,C 180,E1 8155.448,E2 8155.448} C_VEL
LIN {X 0,Y 449.673,Z 532.387,A -85,B 0,C 180,E1 8156.058,E2 8156.058} C_VEL
LIN {X 0,Y 451.745,Z 542.053,A -85,B 0,C 180,E1 8156.535,E2 8156.535} C_VEL
LIN {X 0,Y 452.922,Z 562.419,A -85,B 0,C 180,E1 8157.022,E2 8157.022} C_VEL
LIN {X 0,Y 458.022,Z 579.156,A -85,B 0,C 180,E1 8157.732,E2 8157.732} C_VEL
LIN {X 0,Y 456.078,Z 617.315,A -85,B 0,C 180,E1 8158.999,E2 8158.999} C_VEL
LIN {X 0,Y 453.446,Z 654.27,A -85,B 0,C 180,E1 8161.014,E2 8161.014} C_VEL
LIN {X 0,Y 450.39,Z 687.509,A -85,B 0,C 180,E1 8163.646,E2 8163.646} C_VEL
LIN {X 0,Y 447.493,Z 717.529,A -85,B 0,C 180,E1 8166.921,E2 8166.921} C_VEL
LIN {X 0,Y 445.087,Z 742.636,A -85,B 0,C 180,E1 8170.655,E2 8170.655} C_VEL
LIN {X 0,Y 443.431,Z 762.6,A -85,B 0,C 180,E1 8174.709,E2 8174.709} C_VEL
LIN {X 0,Y 442.474,Z 778.06,A -85,B 0,C 180,E1 8179.19,E2 8179.19} C_VEL
LIN {X 0,Y 442.176,Z 786.873,A -85,B 0,C 180,E1 8183.141,E2 8183.141} C_VEL
LIN {X 0,Y 442.057,Z 790.804,A -85,B 0,C 180,E1 8186.086,E2 8186.086} C_VEL
LIN {X 0,Y 441.984,Z 792.755,A -85,B 0,C 180,E1 8190.001,E2 8190.001} C_VEL
LIN {X 0,Y 442.07,Z 790.884,A -85,B 0,C 180,E1 8193.915,E2 8193.915} C_VEL
LIN {X 0,Y 442.27,Z 784.257,A -85,B 0,C 180,E1 8198.35,E2 8198.35} C_VEL
LIN {X 0,Y 442.783,Z 772.468,A -85,B 0,C 180,E1 8202.799,E2 8202.799} C_VEL
LIN {X 0,Y 444.14,Z 754.636,A -85,B 0,C 180,E1 8207.296,E2 8207.296} C_VEL
LIN {X 0,Y 446.341,Z 732.29,A -85,B 0,C 180,E1 8211.312,E2 8211.312} C_VEL
LIN {X 0,Y 449.399,Z 704.767,A -85,B 0,C 180,E1 8214.967,E2 8214.967} C_VEL
LIN {X 0,Y 452.953,Z 672.216,A -85,B 0,C 180,E1 8218.119,E2 8218.119} C_VEL
LIN {X 0,Y 456.227,Z 637.833,A -85,B 0,C 180,E1 8220.47,E2 8220.47} C_VEL
LIN {X 0,Y 458.923,Z 600.302,A -85,B 0,C 180,E1 8222.169,E2 8222.169} C_VEL
LIN {X 0,Y 459.678,Z 576.716,A -85,B 0,C 180,E1 8222.857,E2 8222.857} C_VEL
LIN {X 0,Y 440.838,Z 529.66,A -85,B 0,C 180,E1 8225.216,E2 8225.216} C_VEL
LIN {X 0,Y 440.735,Z 529.66,A -85,B 0,C 180,E1 8231.133,E2 8231.133} C_VEL
LIN {X 0,Y 440.721,Z 529.66,A -85,B 0,C 180,E1 8236.786,E2 8236.786} C_VEL
LIN {X 0,Y 440.81,Z 529.66,A -85,B 0,C 180,E1 8241.966,E2 8241.966} C_VEL
LIN {X 0,Y 440.762,Z 529.66,A -85,B 0,C 180,E1 8246.789,E2 8246.789} C_VEL
LIN {X 0,Y 440.95,Z 529.66,A -85,B 0,C 180,E1 8253.588,E2 8253.588} C_VEL
LIN {X 0,Y 441.194,Z 529.66,A -85,B 0,C 180,E1 8260.003,E2 8260.003} C_VEL
LIN {X 0,Y 441.219,Z 529.66,A -85,B 0,C 180,E1 8266.152,E2 8266.152} C_VEL
LIN {X 0,Y 441.569,Z 529.66,A -85,B 0,C 180,E1 8272.326,E2 8272.326} C_VEL
LIN {X 0,Y 441.903,Z 529.66,A -85,B 0,C 180,E1 8278.046,E2 8278.046} C_VEL
LIN {X 0,Y 441.744,Z 529.66,A -85,B 0,C 180,E1 8283.92,E2 8283.92} C_VEL
LIN {X 0,Y 441.48,Z 529.66,A -85,B 0,C 180,E1 8289.843,E2 8289.843} C_VEL
LIN {X 0,Y 441.313,Z 529.66,A -85,B 0,C 180,E1 8295.878,E2 8295.878} C_VEL
LIN {X 0,Y 441.046,Z 529.66,A -85,B 0,C 180,E1 8302.513,E2 8302.513} C_VEL
LIN {X 0,Y 440.885,Z 529.66,A -85,B 0,C 180,E1 8308.634,E2 8308.634} C_VEL
LIN {X 0,Y 440.744,Z 529.66,A -85,B 0,C 180,E1 8315.597,E2 8315.597} C_VEL
LIN {X 0,Y 440.874,Z 529.66,A -85,B 0,C 180,E1 8323.064,E2 8323.064} C_VEL
LIN {X 0,Y 450.412,Z 562.608,A -85,B 0,C 180,E1 8324.128,E2 8324.128} C_VEL
LIN {X 0,Y 449.511,Z 630.192,A -85,B 0,C 180,E1 8325.366,E2 8325.366} C_VEL
LIN {X 0,Y 448.254,Z 659.212,A -85,B 0,C 180,E1 8326.695,E2 8326.695} C_VEL
LIN {X 0,Y 446.572,Z 685.184,A -85,B 0,C 180,E1 8328.699,E2 8328.699} C_VEL
LIN {X 0,Y 444.844,Z 707.219,A -85,B 0,C 180,E1 8331.282,E2 8331.282} C_VEL
LIN {X 0,Y 443.515,Z 725.186,A -85,B 0,C 180,E1 8334.406,E2 8334.406} C_VEL
LIN {X 0,Y 442.72,Z 737.758,A -85,B 0,C 180,E1 8337.765,E2 8337.765} C_VEL
LIN {X 0,Y 442.154,Z 745.529,A -85,B 0,C 180,E1 8341.458,E2 8341.458} C_VEL
LIN {X 0,Y 441.848,Z 747.499,A -85,B 0,C 180,E1 8343.641,E2 8343.641} C_VEL
LIN {X 0,Y 441.858,Z 746.794,A -85,B 0,C 180,E1 8347.237,E2 8347.237} C_VEL
LIN {X 0,Y 442.506,Z 740.434,A -85,B 0,C 180,E1 8351.097,E2 8351.097} C_VEL
LIN {X 0,Y 443.177,Z 729.259,A -85,B 0,C 180,E1 8354.527,E2 8354.527} C_VEL
LIN {X 0,Y 444.344,Z 712.735,A -85,B 0,C 180,E1 8357.745,E2 8357.745} C_VEL
LIN {X 0,Y 445.99,Z 691.654,A -85,B 0,C 180,E1 8360.505,E2 8360.505} C_VEL
LIN {X 0,Y 447.662,Z 667.4,A -85,B 0,C 180,E1 8362.642,E2 8362.642} C_VEL
LIN {X 0,Y 449.063,Z 639.929,A -85,B 0,C 180,E1 8364.157,E2 8364.157} C_VEL
LIN {X 0,Y 449.824,Z 609.455,A -85,B 0,C 180,E1 8364.993,E2 8364.993} C_VEL
LIN {X 0,Y 449.467,Z 557.557,A -85,B 0,C 180,E1 8365.881,E2 8365.881} C_VEL
LIN {X 0,Y 441.656,Z 529.66,A -85,B 0,C 180,E1 8366.816,E2 8366.816} C_VEL
LIN {X 0,Y 441.915,Z 529.66,A -85,B 0,C 180,E1 8371.956,E2 8371.956} C_VEL
LIN {X 0,Y 441.555,Z 529.66,A -85,B 0,C 180,E1 8377.856,E2 8377.856} C_VEL
LIN {X 0,Y 441.301,Z 529.66,A -85,B 0,C 180,E1 8383.848,E2 8383.848} C_VEL
LIN {X 0,Y 441.149,Z 529.66,A -85,B 0,C 180,E1 8390.001,E2 8390.001} C_VEL
LIN {X 0,Y 440.9,Z 529.66,A -85,B 0,C 180,E1 8396.418,E2 8396.418} C_VEL
LIN {X 0,Y 440.751,Z 529.66,A -85,B 0,C 180,E1 8403.214,E2 8403.214} C_VEL
LIN {X 0,Y 440.827,Z 529.66,A -85,B 0,C 180,E1 8408.062,E2 8408.062} C_VEL
LIN {X 0,Y 440.697,Z 529.66,A -85,B 0,C 180,E1 8414.02,E2 8414.02} C_VEL
LIN {X 0,Y 440.723,Z 529.66,A -85,B 0,C 180,E1 8419.415,E2 8419.415} C_VEL
LIN {X 0,Y 440.759,Z 529.66,A -85,B 0,C 180,E1 8425.251,E2 8425.251} C_VEL
LIN {X 0,Y 440.878,Z 529.66,A -85,B 0,C 180,E1 8430.014,E2 8430.014} C_VEL
LIN {X 0,Y 456.235,Z 571.724,A -85,B 0,C 180,E1 8432.008,E2 8432.008} C_VEL
LIN {X 0,Y 454.15,Z 606.454,A -85,B 0,C 180,E1 8433.403,E2 8433.403} C_VEL
LIN {X 0,Y 451.512,Z 638.206,A -85,B 0,C 180,E1 8435.436,E2 8435.436} C_VEL
LIN {X 0,Y 448.653,Z 666.804,A -85,B 0,C 180,E1 8438.076,E2 8438.076} C_VEL
LIN {X 0,Y 446.015,Z 692.034,A -85,B 0,C 180,E1 8441.316,E2 8441.316} C_VEL
LIN {X 0,Y 444.007,Z 713.375,A -85,B 0,C 180,E1 8445.142,E2 8445.142} C_VEL
LIN {X 0,Y 442.725,Z 728.965,A -85,B 0,C 180,E1 8449.193,E2 8449.193} C_VEL
LIN {X 0,Y 442.27,Z 738.846,A -85,B 0,C 180,E1 8453.139,E2 8453.139} C_VEL
LIN {X 0,Y 442.109,Z 743.228,A -85,B 0,C 180,E1 8456.083,E2 8456.083} C_VEL
LIN {X 0,Y 442.007,Z 745.329,A -85,B 0,C 180,E1 8459.997,E2 8459.997} C_VEL
LIN {X 0,Y 442.124,Z 743.259,A -85,B 0,C 180,E1 8463.911,E2 8463.911} C_VEL
LIN {X 0,Y 442.47,Z 735.342,A -85,B 0,C 180,E1 8468.508,E2 8468.508} C_VEL
LIN {X 0,Y 443.326,Z 722.083,A -85,B 0,C 180,E1 8472.779,E2 8472.779} C_VEL
LIN {X 0,Y 444.913,Z 703.51,A -85,B 0,C 180,E1 8476.753,E2 8476.753} C_VEL
LIN {X 0,Y 447.262,Z 680.269,A -85,B 0,C 180,E1 8480.229,E2 8480.229} C_VEL
LIN {X 0,Y 449.988,Z 652.493,A -85,B 0,C 180,E1 8483.218,E2 8483.218} C_VEL
LIN {X 0,Y 452.681,Z 621.753,A -85,B 0,C 180,E1 8485.545,E2 8485.545} C_VEL
LIN {X 0,Y 455.006,Z 587.479,A -85,B 0,C 180,E1 8487.267,E2 8487.267} C_VEL
LIN {X 0,Y 455.395,Z 569.451,A -85,B 0,C 180,E1 8487.904,E2 8487.904} C_VEL
LIN {X 0,Y 442.114,Z 533.778,A -85,B 0,C 180,E1 8489.798,E2 8489.798} C_VEL
LIN {X 0,Y 440.924,Z 529.66,A -85,B 0,C 180,E1 8490.071,E2 8490.071} C_VEL
LIN {X 0,Y 440.768,Z 529.66,A -85,B 0,C 180,E1 8495.588,E2 8495.588} C_VEL
LIN {X 0,Y 440.634,Z 529.66,A -85,B 0,C 180,E1 8501.115,E2 8501.115} C_VEL
LIN {X 0,Y 440.7,Z 529.66,A -85,B 0,C 180,E1 8506.78,E2 8506.78} C_VEL
LIN {X 0,Y 440.802,Z 529.66,A -85,B 0,C 180,E1 8511.963,E2 8511.963} C_VEL
LIN {X 0,Y 440.948,Z 530.429,A -85,B 0,C 180,E1 8515.429,E2 8515.429} C_VEL
LIN {X 0,Y 452.922,Z 562.419,A -85,B 0,C 180,E1 8517.022,E2 8517.022} C_VEL
LIN {X 0,Y 453.355,Z 571.333,A -85,B 0,C 180,E1 8517.237,E2 8517.237} C_VEL
LIN {X 0,Y 450.65,Z 585.781,A -85,B 0,C 180,E1 8517.438,E2 8517.438} C_VEL
LIN {X 0,Y 448.37,Z 624.364,A -85,B 0,C 180,E1 8518.898,E2 8518.898} C_VEL
LIN {X 0,Y 445.574,Z 659.691,A -85,B 0,C 180,E1 8521.007,E2 8521.007} C_VEL
LIN {X 0,Y 442.296,Z 693.845,A -85,B 0,C 180,E1 8523.939,E2 8523.939} C_VEL
LIN {X 0,Y 439.322,Z 722.059,A -85,B 0,C 180,E1 8527.269,E2 8527.269} C_VEL
LIN {X 0,Y 436.868,Z 746.715,A -85,B 0,C 180,E1 8531.208,E2 8531.208} C_VEL
LIN {X 0,Y 435.324,Z 765.915,A -85,B 0,C 180,E1 8535.446,E2 8535.446} C_VEL
LIN {X 0,Y 434.509,Z 780.092,A -85,B 0,C 180,E1 8540.001,E2 8540.001} C_VEL
LIN {X 0,Y 434.18,Z 787.98,A -85,B 0,C 180,E1 8544.016,E2 8544.016} C_VEL
LIN {X 0,Y 434.083,Z 791.793,A -85,B 0,C 180,E1 8548.009,E2 8548.009} C_VEL
LIN {X 0,Y 434.208,Z 791.849,A -85,B 0,C 180,E1 8551.992,E2 8551.992} C_VEL
LIN {X 0,Y 434.257,Z 786.592,A -85,B 0,C 180,E1 8556.987,E2 8556.987} C_VEL
LIN {X 0,Y 434.675,Z 776.528,A -85,B 0,C 180,E1 8561.515,E2 8561.515} C_VEL
LIN {X 0,Y 435.941,Z 759.683,A -85,B 0,C 180,E1 8566.335,E2 8566.335} C_VEL
LIN {X 0,Y 438.077,Z 738.423,A -85,B 0,C 180,E1 8570.571,E2 8570.571} C_VEL
LIN {X 0,Y 440.911,Z 713.457,A -85,B 0,C 180,E1 8574.249,E2 8574.249} C_VEL
LIN {X 0,Y 444.475,Z 682.523,A -85,B 0,C 180,E1 8577.612,E2 8577.612} C_VEL
LIN {X 0,Y 447.988,Z 649.13,A -85,B 0,C 180,E1 8580.21,E2 8580.21} C_VEL
LIN {X 0,Y 451.063,Z 612.558,A -85,B 0,C 180,E1 8582.153,E2 8582.153} C_VEL
LIN {X 0,Y 452.435,Z 578.287,A -85,B 0,C 180,E1 8583.302,E2 8583.302} C_VEL
LIN {X 0,Y 432.897,Z 529.66,A -85,B 0,C 180,E1 8585.856,E2 8585.856} C_VEL
LIN {X 0,Y 432.804,Z 529.66,A -85,B 0,C 180,E1 8592.936,E2 8592.936} C_VEL
LIN {X 0,Y 432.805,Z 529.66,A -85,B 0,C 180,E1 8598.518,E2 8598.518} C_VEL
LIN {X 0,Y 432.828,Z 529.66,A -85,B 0,C 180,E1 8603.656,E2 8603.656} C_VEL
LIN {X 0,Y 432.829,Z 529.66,A -85,B 0,C 180,E1 8608.473,E2 8608.473} C_VEL
LIN {X 0,Y 433.061,Z 529.66,A -85,B 0,C 180,E1 8615.286,E2 8615.286} C_VEL
LIN {X 0,Y 433.284,Z 529.66,A -85,B 0,C 180,E1 8621.736,E2 8621.736} C_VEL
LIN {X 0,Y 433.348,Z 529.66,A -85,B 0,C 180,E1 8627.943,E2 8627.943} C_VEL
LIN {X 0,Y 433.735,Z 529.66,A -85,B 0,C 180,E1 8634.012,E2 8634.012} C_VEL
LIN {X 0,Y 433.909,Z 529.66,A -85,B 0,C 180,E1 8640.003,E2 8640.003} C_VEL
LIN {X 0,Y 433.704,Z 529.66,A -85,B 0,C 180,E1 8645.994,E2 8645.994} C_VEL
LIN {X 0,Y 433.447,Z 529.66,A -85,B 0,C 180,E1 8652.89,E2 8652.89} C_VEL
LIN {X 0,Y 433.286,Z 529.66,A -85,B 0,C 180,E1 8658.269,E2 8658.269} C_VEL
LIN {X 0,Y 433.003,Z 529.66,A -85,B 0,C 180,E1 8665.028,E2 8665.028} C_VEL
LIN {X 0,Y 432.813,Z 529.66,A -85,B 0,C 180,E1 8671.534,E2 8671.534} C_VEL
LIN {X 0,Y 432.726,Z 529.66,A -85,B 0,C 180,E1 8676.672,E2 8676.672} C_VEL
LIN {X 0,Y 432.915,Z 529.66,A -85,B 0,C 180,E1 8682.614,E2 8682.614} C_VEL
LIN {X 0,Y 443.012,Z 562.478,A -85,B 0,C 180,E1 8683.753,E2 8683.753} C_VEL
LIN {X 0,Y 442.104,Z 630.193,A -85,B 0,C 180,E1 8685.009,E2 8685.009} C_VEL
LIN {X 0,Y 440.812,Z 658.848,A -85,B 0,C 180,E1 8686.326,E2 8686.326} C_VEL
LIN {X 0,Y 438.987,Z 685.76,A -85,B 0,C 180,E1 8688.427,E2 8688.427} C_VEL
LIN {X 0,Y 437.127,Z 707.908,A -85,B 0,C 180,E1 8691.08,E2 8691.08} C_VEL
LIN {X 0,Y 435.768,Z 725.274,A -85,B 0,C 180,E1 8694.15,E2 8694.15} C_VEL
LIN {X 0,Y 434.83,Z 738.749,A -85,B 0,C 180,E1 8697.841,E2 8697.841} C_VEL
LIN {X 0,Y 434.365,Z 745.191,A -85,B 0,C 180,E1 8700.897,E2 8700.897} C_VEL
LIN {X 0,Y 433.858,Z 748.206,A -85,B 0,C 180,E1 8704.734,E2 8704.734} C_VEL
LIN {X 0,Y 434.232,Z 745.719,A -85,B 0,C 180,E1 8708.599,E2 8708.599} C_VEL
LIN {X 0,Y 434.847,Z 737.535,A -85,B 0,C 180,E1 8712.419,E2 8712.419} C_VEL
LIN {X 0,Y 435.79,Z 723.985,A -85,B 0,C 180,E1 8715.972,E2 8715.972} C_VEL
LIN {X 0,Y 437.3,Z 704.931,A -85,B 0,C 180,E1 8719.192,E2 8719.192} C_VEL
LIN {X 0,Y 439.194,Z 681.226,A -85,B 0,C 180,E1 8721.851,E2 8721.851} C_VEL
LIN {X 0,Y 440.899,Z 655.208,A -85,B 0,C 180,E1 8723.754,E2 8723.754} C_VEL
LIN {X 0,Y 442.096,Z 626.068,A -85,B 0,C 180,E1 8724.981,E2 8724.981} C_VEL
LIN {X 0,Y 442.367,Z 560.05,A -85,B 0,C 180,E1 8726.186,E2 8726.186} C_VEL
LIN {X 0,Y 433.761,Z 529.66,A -85,B 0,C 180,E1 8727.258,E2 8727.258} C_VEL
LIN {X 0,Y 434.003,Z 529.66,A -85,B 0,C 180,E1 8731.992,E2 8731.992} C_VEL
LIN {X 0,Y 433.627,Z 529.66,A -85,B 0,C 180,E1 8738.001,E2 8738.001} C_VEL
LIN {X 0,Y 433.371,Z 529.66,A -85,B 0,C 180,E1 8744.106,E2 8744.106} C_VEL
LIN {X 0,Y 433.218,Z 529.66,A -85,B 0,C 180,E1 8750.384,E2 8750.384} C_VEL
LIN {X 0,Y 432.973,Z 529.66,A -85,B 0,C 180,E1 8756.94,E2 8756.94} C_VEL
LIN {X 0,Y 432.85,Z 529.66,A -85,B 0,C 180,E1 8763.902,E2 8763.902} C_VEL
LIN {X 0,Y 432.782,Z 529.66,A -85,B 0,C 180,E1 8769.904,E2 8769.904} C_VEL
LIN {X 0,Y 432.804,Z 529.66,A -85,B 0,C 180,E1 8775.785,E2 8775.785} C_VEL
LIN {X 0,Y 432.791,Z 529.66,A -85,B 0,C 180,E1 8781.124,E2 8781.124} C_VEL
LIN {X 0,Y 432.785,Z 529.66,A -85,B 0,C 180,E1 8788.463,E2 8788.463} C_VEL
LIN {X 0,Y 432.926,Z 529.914,A -85,B 0,C 180,E1 8789.468,E2 8789.468} C_VEL
LIN {X 0,Y 449.095,Z 573.215,A -85,B 0,C 180,E1 8791.605,E2 8791.605} C_VEL
LIN {X 0,Y 446.835,Z 608.213,A -85,B 0,C 180,E1 8793.06,E2 8793.06} C_VEL
LIN {X 0,Y 443.93,Z 641.041,A -85,B 0,C 180,E1 8795.256,E2 8795.256} C_VEL
